# B&R Automation Studio project GAT (part 8)

#### Configuration.st - not listed in the package file held
```iecst
ACTION ConfigurationInit:

    MachineSettings.DriveConfiguration.PureVirtualAxis.AxisFeatures.FeatureReference.DataAddress := ADR(MachineSettings.AxisFeatures);
    MachineSettings.DriveConfiguration.PureVirtualAxis.AxisFeatures.FeatureReference.NumberOfArrayElements := SIZEOF(MachineSettings.AxisFeatures)/SIZEOF(MachineSettings.AxisFeatures[0]);
    MachineSettings.DriveConfiguration.PureVirtualAxis.AxisFeatures.FeatureReference.NumberOfElements := 0;
    i := 0;
    WHILE ((i <= SIZEOF(MachineSettings.AxisFeatures)/SIZEOF(MachineSettings.AxisFeatures[0])) AND (MachineSettings.AxisFeatures[i] <> '')) DO
        i := i + 1;
    END_WHILE
    MachineSettings.DriveConfiguration.PureVirtualAxis.AxisFeatures.FeatureReference.NumberOfElements := i;

    MC_BR_ProcessConfig_AX.DataAddress := ADR(MachineSettings.BaseConfiguration);
    MC_BR_ProcessConfig_AX.DataType := mcCFG_AX;

    MC_BR_ProcessConfig_ACP.DataAddress := ADR(MachineSettings.DriveConfiguration);
    MC_BR_ProcessConfig_ACP.DataType := mcCFG_PURE_V_AX;

    configurationState := CONFIG_STATE_INIT;

END_ACTION

ACTION Configuration:

    CASE configurationState OF
        CONFIG_STATE_INIT:

            (* build up the string for the name *)
            MC_BR_ProcessConfig_ACP.Name := MpAxisBasicFB.Info.HardwareInfo.Axis.ConfigElementLocation;
            MC_BR_ProcessConfig_AX.Name := MpAxisBasicFB.Info.HardwareInfo.Axis.AxisName;

            IF (MpAxisBasicFB.Active = TRUE) THEN
                configurationState := CONFIG_STATE_READ;
            END_IF

        CONFIG_STATE_READ:
            MC_BR_ProcessConfig_ACP.Mode := mcPCM_LOAD;
            MC_BR_ProcessConfig_ACP.Execute := TRUE;

            MC_BR_ProcessConfig_AX.Mode := mcPCM_LOAD;
            MC_BR_ProcessConfig_AX.Execute := TRUE;
            IF (MC_BR_ProcessConfig_ACP.Done = TRUE) AND (MC_BR_ProcessConfig_AX.Done = TRUE) THEN
                MC_BR_ProcessConfig_ACP.Execute := FALSE;
                MC_BR_ProcessConfig_AX.Execute := FALSE;
                configurationState := CONFIG_STATE_READY;
            END_IF

        CONFIG_STATE_WRITE:
            MC_BR_ProcessConfig_ACP.Mode := mcPCM_SAVE;
            MC_BR_ProcessConfig_ACP.Execute := TRUE;

            MC_BR_ProcessConfig_AX.Mode := mcPCM_SAVE;
            MC_BR_ProcessConfig_AX.Execute := TRUE;
            IF (MC_BR_ProcessConfig_ACP.Done = TRUE) AND (MC_BR_ProcessConfig_AX.Done = TRUE) THEN
                MC_BR_ProcessConfig_ACP.Execute := FALSE;
                MC_BR_ProcessConfig_AX.Execute := FALSE;
                configurationState := CONFIG_STATE_READY;
            END_IF

        CONFIG_STATE_READY:

    END_CASE

    MC_BR_ProcessConfig_ACP();
    MC_BR_ProcessConfig_AX();

END_ACTION
```

#### Main.st - not listed in the package file held
```iecst
(***********************************************************************************************************************
* Copyright: B&R Industrial Automation GmbH
* Description: This program implements an axis control
***********************************************************************************************************************)

PROGRAM _INIT

    ST_name(0, ADR(AxisControl.Status.TaskName), 0);

    MpAlarmXCoreFB.Enable := TRUE;
    ConfigurationInit;

    MpAxisBasicFB.Enable := TRUE;
    MpAxisBasicFB.MpLink := ADR(gAxisTest);

    AxisInit;

END_PROGRAM

PROGRAM _CYCLIC

    MpAxisBasicFB.MpLink := ADR(gAxisTest);
    MC_BR_CheckRestorePositionDataFB.Axis := ADR(gAxisTest);

    SimulationControl;
    AxisStateMachine;
    AxisCyclic;
    RecipeCyclic;

    MpAlarmXCoreFB.MpLink := ADR(gAlarmXCore_Test);
    MpAlarmXCoreFB();

END_PROGRAM

PROGRAM _EXIT

    MpRecipeRegPar_MachineFB.Enable := FALSE;
    MpRecipeRegPar_MachineFB();

    MpRecipeRegPar_UserFB.Enable := FALSE;
    MpRecipeRegPar_UserFB();

    MpRecipeRegPar_PreFB.Enable := FALSE;
    MpRecipeRegPar_PreFB();

    MpRecipeRegPar_UserPreFB.Enable := FALSE;
    MpRecipeRegPar_UserPreFB();

    MpAxisBasicFB.Enable := FALSE;
    MpAxisBasicFB();

    MpAlarmXCoreFB.Enable := FALSE;
    MpAlarmXCoreFB();

END_PROGRAM
```

### Program Logical/Infrastructure/UsbDevLink/UsbDevLink (IEC)

#### UsbDevLink.st - Init, cyclic, exit code
```iecst
//*********************************************************************************
//* Copyright: B&R Industrial Automation GmbH
//* Author:    MITC
//* Created:   September 26, 2021/09:19
//* This task shall automatically detect and (un)link USB storage devices
//*********************************************************************************

PROGRAM _INIT
	DevLinkCtrl.FUB.DevLink_0.enable := FALSE;
	DevLinkCtrl.FUB.DevUnlink_0.enable := FALSE;
	DevLinkCtrl.FUB.UsbNodeGet_0.enable := FALSE;
	DevLinkCtrl.FUB.UsbNodeListGet_0.enable := FALSE;
	DevLinkCtrl.FUB.DevLink_0();
	DevLinkCtrl.FUB.DevUnlink_0();
	DevLinkCtrl.FUB.UsbNodeGet_0();
	DevLinkCtrl.FUB.UsbNodeListGet_0();

	FOR Index := 0 TO MAX_IDX_USB_DEV_LIST DO
		AttachedUSB[Index] := FALSE;
		gUSBAvailable[Index] := FALSE;
	END_FOR
END_PROGRAM

PROGRAM _CYCLIC
	// BEGIN OF STATE MACHINE
	CASE DevLinkCtrl.Step OF
		// WAIT STEP
		STATE_WAIT:
			// UPDATE USB INFO LIST IF THE NODE LIST HAS CHANGED
			IF (brsmemcmp(ADR(DevLinkCtrl.Params.NodeList), ADR(LastNodeList), SIZEOF(LastNodeList)) <> 0) THEN
				DevLinkCtrl.Cmd.GetUSBInfo := TRUE;
				// preserve the previously created drive information in CASE the order has changed when unplugging a device
				FOR DevLinkCtrl.Params.Index := 0 TO MAX_IDX_USB_DEV_LIST DO
					FOR Index := 0 TO MAX_IDX_USB_DEV_LIST DO
						IF ((DevLinkCtrl.Params.NodeList[DevLinkCtrl.Params.Index] = LastNodeList[Index]) AND
							(DevLinkCtrl.Params.Index <> Index) AND (LastNodeList[Index] <> 0)) THEN
							brsmemcpy(ADR(TempUSBInfo), ADR(DevLinkCtrl.Params.NodeInfoList[DevLinkCtrl.Params.Index]), SIZEOF(TempUSBInfo));
							brsmemcpy(ADR(DevLinkCtrl.Params.NodeInfoList[DevLinkCtrl.Params.Index]), ADR(DevLinkCtrl.Params.NodeInfoList[Index]), SIZEOF(TempUSBInfo));
							brsmemcpy(ADR(DevLinkCtrl.Params.NodeInfoList[Index]), ADR(TempUSBInfo), SIZEOF(TempUSBInfo));
							brsmemcpy(ADR(TempFileDevName), ADR(DevLinkCtrl.Params.FileDevName[DevLinkCtrl.Params.Index]), SIZEOF(TempFileDevName));
							brsmemcpy(ADR(DevLinkCtrl.Params.FileDevName[DevLinkCtrl.Params.Index]), ADR(DevLinkCtrl.Params.FileDevName[Index]), SIZEOF(TempFileDevName));
							brsmemcpy(ADR(DevLinkCtrl.Params.FileDevName[Index]), ADR(TempFileDevName), SIZEOF(TempFileDevName));
							TempFileDevHandle := DevLinkCtrl.Params.FileDevHandle[DevLinkCtrl.Params.Index];
							DevLinkCtrl.Params.FileDevHandle[DevLinkCtrl.Params.Index] := DevLinkCtrl.Params.FileDevHandle[Index];
							DevLinkCtrl.Params.FileDevHandle[Index] := TempFileDevHandle;
						END_IF
					END_FOR
				END_FOR
				brsmemcpy(ADR(LastNodeList), ADR(DevLinkCtrl.Params.NodeList), SIZEOF(LastNodeList));
			END_IF

			FOR DevLinkCtrl.Params.Index := 0 TO MAX_IDX_USB_DEV_LIST DO
				// SKIP IF LOADING USB LIST INFORMATION
				IF DevLinkCtrl.Cmd.GetUSBInfo THEN
					EXIT;
				END_IF
				// ALWAYS KEEP DEVICES LINKED WHEN AVAILABLE
				IF ((DevLinkCtrl.Params.FileDevHandle[DevLinkCtrl.Params.Index] = 0) AND AttachedUSB[DevLinkCtrl.Params.Index]
					AND (DevLinkCtrl.Params.NodeList[DevLinkCtrl.Params.Index] <> 0)) THEN
					DevLinkCtrl.Cmd.DevLink := TRUE;
					EXIT;
				END_IF
				// UNLINK DEVICE IF IT IS NOT CONNECTED ANYMORE
				IF ((DevLinkCtrl.Params.FileDevHandle[DevLinkCtrl.Params.Index] <> 0) AND
					(DevLinkCtrl.Params.NodeInfoList[DevLinkCtrl.Params.Index].interfaceClass <> 8)) THEN
					DevLinkCtrl.Cmd.DevUnlink := TRUE;
					EXIT;
				END_IF
			END_FOR

			// CHECK FOR USB DEVICES EVERY 3 SEC
			TON_0.PT := t#3s;
			IF (TON_0.Q AND NOT DevLinkCtrl.Cmd.GetUSBInfo AND NOT DevLinkCtrl.Cmd.DevLink AND NOT DevLinkCtrl.Cmd.DevUnlink) THEN
				DevLinkCtrl.Cmd.GetUSBList := TRUE;
				TON_0.IN := FALSE;
			ELSE
				TON_0.IN := TRUE;
			END_IF
			TON_0();

			IF DevLinkCtrl.Cmd.GetUSBInfo THEN
				// get usb info cmd
				DevLinkCtrl.Cmd.GetUSBInfo := FALSE;
				brsmemset(ADR(DevLinkCtrl.Params.NodeInfoList), 0, SIZEOF(DevLinkCtrl.Params.NodeInfoList));
				DevLinkCtrl.Step := STATE_GET_USB_INFO;
				DevLinkCtrl.Params.Index := 0;
			ELSIF DevLinkCtrl.Cmd.GetUSBList THEN
				// get usb list cmd
				DevLinkCtrl.Cmd.GetUSBList := FALSE;
				brsmemset(ADR(DevLinkCtrl.Params.NodeList), 0, SIZEOF(DevLinkCtrl.Params.NodeList));
				DevLinkCtrl.Step := STATE_GET_USB_LIST;
			ELSIF DevLinkCtrl.Cmd.DevLink THEN
				// link cmd
				DevLinkCtrl.Cmd.DevLink := FALSE;
				DevLinkCtrl.Step := STATE_DEV_LINK;
			ELSIF DevLinkCtrl.Cmd.DevUnlink THEN
				// unlink cmd
				DevLinkCtrl.Cmd.DevUnlink := FALSE;
				DevLinkCtrl.Step := STATE_DEV_UNLINK;
			END_IF
			// END OF WAIT STEP

			// GET USB LIST STEP
		STATE_GET_USB_LIST:
			// SET FUB PARAMS
			DevLinkCtrl.FUB.UsbNodeListGet_0.enable := TRUE;
			DevLinkCtrl.FUB.UsbNodeListGet_0.bufferSize := SIZEOF(DevLinkCtrl.Params.NodeList);
			DevLinkCtrl.FUB.UsbNodeListGet_0.pBuffer := ADR(DevLinkCtrl.Params.NodeList);

			// ERROR HANDLING
			IF ((DevLinkCtrl.FUB.UsbNodeListGet_0.status = ERR_OK) OR (DevLinkCtrl.FUB.UsbNodeListGet_0.status = asusbERR_USB_NOTFOUND)) THEN
				DevLinkCtrl.Step := STATE_WAIT;
				DevLinkCtrl.FUB.UsbNodeListGet_0.enable := FALSE;
			ELSIF ((DevLinkCtrl.FUB.UsbNodeListGet_0.status <> ERR_FUB_BUSY) AND (DevLinkCtrl.FUB.UsbNodeListGet_0.status <> ERR_FUB_ENABLE_FALSE)
				AND (DevLinkCtrl.FUB.UsbNodeListGet_0.status <> asusbERR_USB_NOTFOUND)) THEN
				DevLinkCtrl.Step := STATE_ERROR_USB;
				DevLinkCtrl.Params.ErrorID := DevLinkCtrl.FUB.UsbNodeListGet_0.status;
				DevLinkCtrl.FUB.UsbNodeListGet_0.enable := FALSE;
			END_IF
			// CALL OF FUB
			DevLinkCtrl.FUB.UsbNodeListGet_0();
			// END OF GET USB LIST STEP

			// GET USB INFO STEP
		STATE_GET_USB_INFO:
			// SET FUB PARAMS
			DevLinkCtrl.FUB.UsbNodeGet_0.bufferSize := SIZEOF(DevLinkCtrl.Params.NodeInfoList[DevLinkCtrl.Params.Index]);
			DevLinkCtrl.FUB.UsbNodeGet_0.enable := TRUE;
			DevLinkCtrl.FUB.UsbNodeGet_0.nodeId := DevLinkCtrl.Params.NodeList[DevLinkCtrl.Params.Index];
			DevLinkCtrl.FUB.UsbNodeGet_0.pBuffer := ADR(DevLinkCtrl.Params.NodeInfoList[DevLinkCtrl.Params.Index]);

			// CHECK IF DevLinkCtrl.Params.Index CONTAINS AN ENTRY
			IF (DevLinkCtrl.Params.NodeList[DevLinkCtrl.Params.Index] = 0) THEN
				DevLinkCtrl.FUB.UsbNodeGet_0.enable := TRUE;
				brsmemset(ADR(DevLinkCtrl.Params.NodeInfoList[DevLinkCtrl.Params.Index]), 0, SIZEOF(DevLinkCtrl.Params.NodeInfoList[DevLinkCtrl.Params.Index]));
				DevLinkCtrl.Params.Index := DevLinkCtrl.Params.Index + 1;
			END_IF

			// ERROR HANDLING
			IF (DevLinkCtrl.FUB.UsbNodeGet_0.status = ERR_OK) THEN
				DevLinkCtrl.FUB.UsbNodeGet_0.enable := FALSE;
				DevLinkCtrl.Params.Index := DevLinkCtrl.Params.Index + 1;
			ELSIF ((DevLinkCtrl.FUB.UsbNodeGet_0.status <> ERR_FUB_BUSY) AND (DevLinkCtrl.FUB.UsbNodeGet_0.status <> ERR_FUB_ENABLE_FALSE)) THEN
				DevLinkCtrl.Step := STATE_ERROR_USB;
				DevLinkCtrl.Params.ErrorID := DevLinkCtrl.FUB.UsbNodeGet_0.status;
				DevLinkCtrl.FUB.UsbNodeGet_0.enable := FALSE;
			END_IF

			// END OF LIST REACHED
			IF (DevLinkCtrl.Params.Index > MAX_IDX_USB_DEV_LIST) THEN
				DevLinkCtrl.FUB.UsbNodeGet_0.enable := FALSE;
				DevLinkCtrl.Step := STATE_WAIT;
				FOR DevLinkCtrl.Params.Index := 0 TO MAX_IDX_USB_DEV_LIST DO
					IF (DevLinkCtrl.Params.NodeInfoList[DevLinkCtrl.Params.Index].interfaceClass = 8) THEN
						AttachedUSB[DevLinkCtrl.Params.Index] := TRUE;
					ELSE
						AttachedUSB[DevLinkCtrl.Params.Index] := FALSE;
						gUSBAvailable[DevLinkCtrl.Params.Index] := FALSE;
					END_IF
				END_FOR
			END_IF

			// CALL OF FUB
			DevLinkCtrl.FUB.UsbNodeGet_0();
			// END OF GET USB INFO STEP

			// LINK DEVICE STEP
		STATE_DEV_LINK:
            // SET FUB PARAMS
			DevLinkCtrl.FUB.DevLink_0.enable := TRUE;
			DevLinkCtrl.FUB.DevLink_0.pDevice := ADR(DevLinkCtrl.Params.FileDevName[DevLinkCtrl.Params.Index]);
			brsstrcpy(ADR(DevLinkCtrl.Params.LinkParam), ADR('/DEVICE='));
			brsstrcat(ADR(DevLinkCtrl.Params.LinkParam), ADR(DevLinkCtrl.Params.NodeInfoList[DevLinkCtrl.Params.Index].ifName));
			DevLinkCtrl.FUB.DevLink_0.pParam := ADR(DevLinkCtrl.Params.LinkParam);

			// ERROR HANDLING
			IF (DevLinkCtrl.FUB.DevLink_0.status = ERR_OK) THEN
				DevLinkCtrl.Params.FileDevHandle[DevLinkCtrl.Params.Index] := DevLinkCtrl.FUB.DevLink_0.handle;
				DevLinkCtrl.Step := STATE_WAIT;
				DevLinkCtrl.FUB.DevLink_0.enable := FALSE;
				FOR Index := 0 TO MAX_IDX_USB_DEV_LIST DO
					gUSBAvailable[Index] := AttachedUSB[Index];
				END_FOR
			ELSIF ((DevLinkCtrl.FUB.DevLink_0.status <> ERR_FUB_BUSY) AND (DevLinkCtrl.FUB.DevLink_0.status <> ERR_FUB_ENABLE_FALSE)) THEN
				DevLinkCtrl.Step := STATE_ERROR_USB;
				DevLinkCtrl.Params.ErrorID := DevLinkCtrl.FUB.DevLink_0.status;
				DevLinkCtrl.FUB.DevLink_0.enable := FALSE;
			END_IF
			// CALL OF FUB
			DevLinkCtrl.FUB.DevLink_0();
			// END OF LINK DEVICE STEP

			// UNLINK DEVICE STEP
		STATE_DEV_UNLINK:
			// SET FUB PARAMS
			DevLinkCtrl.FUB.DevUnlink_0.enable := TRUE;
			DevLinkCtrl.FUB.DevUnlink_0.handle := DevLinkCtrl.Params.FileDevHandle[DevLinkCtrl.Params.Index];

			// CHECK IF WE HAVE A HANDLE
			IF (DevLinkCtrl.Params.FileDevHandle[DevLinkCtrl.Params.Index] = 0) THEN
				DevLinkCtrl.FUB.DevUnlink_0.enable := FALSE;
				DevLinkCtrl.Step := STATE_WAIT;
			END_IF

			// ERROR HANDLING
			IF (DevLinkCtrl.FUB.DevUnlink_0.status = ERR_OK) THEN
				DevLinkCtrl.Params.FileDevHandle[DevLinkCtrl.Params.Index] := 0;
				DevLinkCtrl.FUB.DevUnlink_0.enable := FALSE;
				DevLinkCtrl.Step := STATE_WAIT;
			ELSIF ((DevLinkCtrl.FUB.DevUnlink_0.status <> ERR_FUB_BUSY) AND (DevLinkCtrl.FUB.DevUnlink_0.status <> ERR_FUB_ENABLE_FALSE)) THEN
				DevLinkCtrl.Step := STATE_ERROR_USB;
				DevLinkCtrl.Params.ErrorID := DevLinkCtrl.FUB.DevUnlink_0.status;
				DevLinkCtrl.FUB.DevUnlink_0.enable := FALSE;
			END_IF
			// CALL OF FUB
			DevLinkCtrl.FUB.DevUnlink_0();
			// END OF UNLINK DEVICE STEP

			// WAIT FOR ERRACK CMD STEP
		STATE_ERROR_USB:
			// DELETE ERROR ID AND GO BACK TO WAIT STEP WHEN ERROR IS ACKNOWLEDGED
			IF DevLinkCtrl.Cmd.ErrAck THEN
				DevLinkCtrl.Params.ErrorID := 0;
				DevLinkCtrl.Cmd.ErrAck := FALSE;
				DevLinkCtrl.Step := STATE_WAIT;
			END_IF
		// END OF WAIT FOR ERRACK STEP
	END_CASE;
	// END OF STATE MACHINE
END_PROGRAM

PROGRAM _EXIT
	// Insert code here
END_PROGRAM
```

#### UsbDevLink.var - Local variables
```iecst
(*********************************************************************************
 * Copyright: Bernecker + Rainer
 * Author:    deermannd
 * Created:   21 October, 2015/1:30 PM
 *********************************************************************************
 * DevLinkTask variables of project
 *********************************************************************************)
VAR
	DevLinkCtrl : DevLinkCtrlType := (Params:=(FileDevName:=['USB1','USB2'])); (*DevLink Control variable*)
	TON_0 : TON; (*timer to refresh available usb devices*)
	LastNodeList : ARRAY[0..MAX_IDX_USB_DEV_LIST] OF UDINT; (*temp variable to check if the node list has changed*)
	TempFileDevHandle : UDINT := 0;
	TempFileDevName : STRING[30] := '';
	TempUSBInfo : usbNode_typ := (0); (*temp info structure*)
	Index : USINT := 0; (*index to loop through ussb devices*)
	AttachedUSB : ARRAY[0..MAX_IDX_USB_DEV_LIST] OF BOOL := [2(FALSE)];
END_VAR
```

#### Types.typ - not listed in the package file held
```iecst
(*********************************************************************************
 * Copyright: Bernecker + Rainer
 * Author:    MITC
 * Created:   21 October, 2015/1:30 PM
 *********************************************************************************
 * DevLinkTask data types of project
 *********************************************************************************)

TYPE
	StepType :
		( (*enumeration of the possible machine states*)
		STATE_WAIT := 0, (*waiting for cmds*)
		STATE_GET_USB_LIST, (*getting list of usb devices*)
		STATE_GET_USB_INFO, (*getting info from a usb device*)
		STATE_DEV_LINK, (*linking device*)
		STATE_DEV_UNLINK, (*unlinking device*)
		STATE_ERROR_USB (*some FUB returned an error*)
		);
	CommandType : 	STRUCT  (*possible machine cmds*)
		GetUSBList : BOOL; (*get usb list cmd*)
		GetUSBInfo : BOOL; (*get usb info cmd*)
		DevLink : BOOL; (*link cmd*)
		DevUnlink : BOOL; (*unlink cmd*)
		ErrAck : BOOL; (*error acknowledge cmd*)
	END_STRUCT;
	DevLink_FUB_Type : 	STRUCT  (*contains all needed FileIO FUBs*)
		UsbNodeListGet_0 : UsbNodeListGet;
		UsbNodeGet_0 : UsbNodeGet;
		UsbMsDeviceReady_0 : UsbMsDeviceReady;
		DevLink_0 : DevLink;
		DevUnlink_0 : DevUnlink;
	END_STRUCT;
	DevLinkCtrlType : 	STRUCT  (*Control structure which contains everything necessary for the file handling machine*)
		Step : StepType; (*actual step*)
		Cmd : CommandType; (*when in STATE_WAIT a cmd with value true will change the machine state*)
		FUB : DevLink_FUB_Type; (*all DevLink FUBs*)
		Params : ParamsType; (*parameters like file device, error ID, Buffer, ...*)
	END_STRUCT;
	ParamsType : 	STRUCT  (*Parameter structure*)
		ErrorID : UINT; (*the error id from a FUB is stored here in case of error*)
		NodeList : ARRAY[0..MAX_IDX_USB_DEV_LIST]OF UDINT; (*List of connected usb devices*)
		NodeInfoList : ARRAY[0..MAX_IDX_USB_DEV_LIST]OF usbNode_typ; (*Buffer for usb info*)
		FileDevName : ARRAY[0..MAX_IDX_USB_DEV_LIST]OF STRING[30]; (*file device names*)
		FileDevHandle : ARRAY[0..MAX_IDX_USB_DEV_LIST]OF UDINT; (*needed for unlinking the device again*)
		LinkParam : STRING[30]; (*param string to link a device*)
		Index : USINT; (*list index*)
	END_STRUCT;
END_TYPE
```

#### Variables.var - not listed in the package file held
```iecst
(*********************************************************************************
 * Copyright: Bernecker + Rainer
 * Author:    deermannd
 * Created:   21 October, 2015/1:30 PM
 *********************************************************************************
 * DevLinkTask variables of project
 *********************************************************************************)
VAR CONSTANT
	MAX_IDX_USB_DEV_LIST : USINT := 1; (*Max index for usb storage devices (1 means up to two devices with index 0 and 1)*)
END_VAR
VAR
	DevLinkCtrl : DevLinkCtrlType := (Params:=(FileDevName:=['USB1','USB2'])); (*DevLink Control variable*)
	TON_0 : TON; (*timer to refresh available usb devices*)
	LastNodeList : ARRAY[0..MAX_IDX_USB_DEV_LIST] OF UDINT; (*temp variable to check if the node list has changed*)
	TempFileDevHandle : UDINT := 0;
	TempFileDevName : STRING[30] := '';
	TempUSBInfo : usbNode_typ := (0); (*temp info structure*)
	Index : USINT := 0; (*index to loop through ussb devices*)
	bAttachedUSB : ARRAY[0..MAX_IDX_USB_DEV_LIST] OF BOOL := [2(FALSE)];
END_VAR
```

#### Main.st - not listed in the package file held
```iecst
(*********************************************************************************
 * Copyright: B&R Industrial Automation GmbH
 * Author:    MITC
 * Created:   September 26, 2021/09:19
 * This task shall automatically detect and (un)link USB storage devices
 *********************************************************************************)

PROGRAM _INIT
	DevLinkCtrl.FUB.DevLink_0.enable		:= FALSE;
	DevLinkCtrl.FUB.DevUnlink_0.enable 		:= FALSE;
	DevLinkCtrl.FUB.UsbNodeGet_0.enable		:= FALSE;
	DevLinkCtrl.FUB.UsbNodeListGet_0.enable	:= FALSE;
	DevLinkCtrl.FUB.DevLink_0();
	DevLinkCtrl.FUB.DevUnlink_0();
	DevLinkCtrl.FUB.UsbNodeGet_0();
	DevLinkCtrl.FUB.UsbNodeListGet_0();

	FOR Index := 0 TO MAX_IDX_USB_DEV_LIST DO
		bAttachedUSB[Index] 				:= FALSE;
		gbUSBAvail[Index]					:= FALSE;
	END_FOR;
END_PROGRAM

PROGRAM _CYCLIC
	(* BEGIN OF STATE MACHINE *)
	CASE DevLinkCtrl.Step OF
		(* WAIT STEP *)
		STATE_WAIT:
			(* UPDATE USB INFO LIST IF THE NODE LIST HAS CHANGED *)
			IF (brsmemcmp(ADR(DevLinkCtrl.Params.NodeList), ADR(LastNodeList), SIZEOF(LastNodeList)) <> 0) THEN
				DevLinkCtrl.Cmd.GetUSBInfo		:= TRUE;
				(* preserve the previously created drive information in CASE the order has changed when unplugging a device *)
				FOR DevLinkCtrl.Params.Index := 0 TO MAX_IDX_USB_DEV_LIST DO
					FOR Index := 0 TO MAX_IDX_USB_DEV_LIST DO
						IF ((DevLinkCtrl.Params.NodeList[DevLinkCtrl.Params.Index] = LastNodeList[Index]) AND
							(DevLinkCtrl.Params.Index <> Index) AND (LastNodeList[Index] <> 0)) THEN
							brsmemcpy(ADR(TempUSBInfo), ADR(DevLinkCtrl.Params.NodeInfoList[DevLinkCtrl.Params.Index]), SIZEOF(TempUSBInfo));
							brsmemcpy(ADR(DevLinkCtrl.Params.NodeInfoList[DevLinkCtrl.Params.Index]), ADR(DevLinkCtrl.Params.NodeInfoList[Index]), SIZEOF(TempUSBInfo));
							brsmemcpy(ADR(DevLinkCtrl.Params.NodeInfoList[Index]), ADR(TempUSBInfo), SIZEOF(TempUSBInfo));
							brsmemcpy(ADR(TempFileDevName), ADR(DevLinkCtrl.Params.FileDevName[DevLinkCtrl.Params.Index]), SIZEOF(TempFileDevName));
							brsmemcpy(ADR(DevLinkCtrl.Params.FileDevName[DevLinkCtrl.Params.Index]), ADR(DevLinkCtrl.Params.FileDevName[Index]), SIZEOF(TempFileDevName));
							brsmemcpy(ADR(DevLinkCtrl.Params.FileDevName[Index]), ADR(TempFileDevName), SIZEOF(TempFileDevName));
							TempFileDevHandle											:= DevLinkCtrl.Params.FileDevHandle[DevLinkCtrl.Params.Index];
							DevLinkCtrl.Params.FileDevHandle[DevLinkCtrl.Params.Index]	:= DevLinkCtrl.Params.FileDevHandle[Index];
							DevLinkCtrl.Params.FileDevHandle[Index]						:= TempFileDevHandle;
						END_IF;
					END_FOR;
				END_FOR;
				brsmemcpy(ADR(LastNodeList), ADR(DevLinkCtrl.Params.NodeList), SIZEOF(LastNodeList));
			END_IF;

			FOR DevLinkCtrl.Params.Index := 0 TO MAX_IDX_USB_DEV_LIST DO
				(* SKIP IF LOADING USB LIST INFORMATION *)
				IF DevLinkCtrl.Cmd.GetUSBInfo THEN
					EXIT;
				END_IF;
				(* ALWAYS KEEP DEVICES LINKED WHEN AVAILABLE *)
				IF ((DevLinkCtrl.Params.FileDevHandle[DevLinkCtrl.Params.Index] = 0) AND bAttachedUSB[DevLinkCtrl.Params.Index]
					AND (DevLinkCtrl.Params.NodeList[DevLinkCtrl.Params.Index] <> 0)) THEN
					DevLinkCtrl.Cmd.DevLink		:= TRUE;
					EXIT;
				END_IF;
				(* UNLINK DEVICE IF IT IS NOT CONNECTED ANYMORE *)
				IF ((DevLinkCtrl.Params.FileDevHandle[DevLinkCtrl.Params.Index] <> 0) AND
					(DevLinkCtrl.Params.NodeInfoList[DevLinkCtrl.Params.Index].interfaceClass <> 8)) THEN
					DevLinkCtrl.Cmd.DevUnlink	:= TRUE;
					EXIT;
				END_IF;
			END_FOR;

			(* CHECK FOR USB DEVICES EVERY 3 SEC *)
			TON_0.PT							:= t#3s;
			IF (TON_0.Q AND NOT DevLinkCtrl.Cmd.GetUSBInfo AND NOT DevLinkCtrl.Cmd.DevLink AND NOT DevLinkCtrl.Cmd.DevUnlink) THEN
				DevLinkCtrl.Cmd.GetUSBList		:= TRUE;
				TON_0.IN						:= FALSE;
			ELSE
				TON_0.IN						:= TRUE;
			END_IF;
			TON_0();

			IF DevLinkCtrl.Cmd.GetUSBInfo THEN
				(* get usb info cmd *)
				DevLinkCtrl.Cmd.GetUSBInfo	:= FALSE;
				brsmemset(ADR(DevLinkCtrl.Params.NodeInfoList), 0, SIZEOF(DevLinkCtrl.Params.NodeInfoList));
				DevLinkCtrl.Step			:= STATE_GET_USB_INFO;
				DevLinkCtrl.Params.Index	:= 0;
			ELSIF DevLinkCtrl.Cmd.GetUSBList THEN
				(* get usb list cmd *)
				DevLinkCtrl.Cmd.GetUSBList	:= FALSE;
				brsmemset(ADR(DevLinkCtrl.Params.NodeList), 0, SIZEOF(DevLinkCtrl.Params.NodeList));
				DevLinkCtrl.Step			:= STATE_GET_USB_LIST;
			ELSIF DevLinkCtrl.Cmd.DevLink THEN
				(* link cmd *)
				DevLinkCtrl.Cmd.DevLink		:= FALSE;
				DevLinkCtrl.Step			:= STATE_DEV_LINK;
			ELSIF DevLinkCtrl.Cmd.DevUnlink THEN
				(* unlink cmd *)
				DevLinkCtrl.Cmd.DevUnlink	:= FALSE;
				DevLinkCtrl.Step			:= STATE_DEV_UNLINK;
			END_IF;
			(* END OF WAIT STEP *)

			(* GET USB LIST STEP *)
		STATE_GET_USB_LIST:
			(* SET FUB PARAMS *)
			DevLinkCtrl.FUB.UsbNodeListGet_0.enable		:= TRUE;
			DevLinkCtrl.FUB.UsbNodeListGet_0.bufferSize	:= SIZEOF(DevLinkCtrl.Params.NodeList);
			DevLinkCtrl.FUB.UsbNodeListGet_0.pBuffer	:= ADR(DevLinkCtrl.Params.NodeList);

			(* ERROR HANDLING *)
			IF ((DevLinkCtrl.FUB.UsbNodeListGet_0.status = ERR_OK) OR (DevLinkCtrl.FUB.UsbNodeListGet_0.status = asusbERR_USB_NOTFOUND)) THEN
				DevLinkCtrl.Step						:= STATE_WAIT;
				DevLinkCtrl.FUB.UsbNodeListGet_0.enable	:= FALSE;
			ELSIF ((DevLinkCtrl.FUB.UsbNodeListGet_0.status <> ERR_FUB_BUSY) AND (DevLinkCtrl.FUB.UsbNodeListGet_0.status <> ERR_FUB_ENABLE_FALSE)
				AND (DevLinkCtrl.FUB.UsbNodeListGet_0.status <> asusbERR_USB_NOTFOUND)) THEN
				DevLinkCtrl.Step						:= STATE_ERROR_USB;
				DevLinkCtrl.Params.ErrorID				:= DevLinkCtrl.FUB.UsbNodeListGet_0.status;
				DevLinkCtrl.FUB.UsbNodeListGet_0.enable	:= FALSE;
			END_IF;
			(* CALL OF FUB *)
			DevLinkCtrl.FUB.UsbNodeListGet_0();
			(* END OF GET USB LIST STEP *)

			(* GET USB INFO STEP *)
		STATE_GET_USB_INFO:
			(* SET FUB PARAMS *)
			DevLinkCtrl.FUB.UsbNodeGet_0.bufferSize	:= SIZEOF(DevLinkCtrl.Params.NodeInfoList[DevLinkCtrl.Params.Index]);
			DevLinkCtrl.FUB.UsbNodeGet_0.enable		:= TRUE;
			DevLinkCtrl.FUB.UsbNodeGet_0.nodeId		:= DevLinkCtrl.Params.NodeList[DevLinkCtrl.Params.Index];
			DevLinkCtrl.FUB.UsbNodeGet_0.pBuffer	:= ADR(DevLinkCtrl.Params.NodeInfoList[DevLinkCtrl.Params.Index]);

			(* CHECK IF DevLinkCtrl.Params.Index CONTAINS AN ENTRY *)
			IF (DevLinkCtrl.Params.NodeList[DevLinkCtrl.Params.Index] = 0) THEN
				DevLinkCtrl.FUB.UsbNodeGet_0.enable	:= TRUE;
				brsmemset(ADR(DevLinkCtrl.Params.NodeInfoList[DevLinkCtrl.Params.Index]), 0, SIZEOF(DevLinkCtrl.Params.NodeInfoList[DevLinkCtrl.Params.Index]));
				DevLinkCtrl.Params.Index			:= DevLinkCtrl.Params.Index + 1;
			END_IF;

			(* ERROR HANDLING *)
			IF (DevLinkCtrl.FUB.UsbNodeGet_0.status = ERR_OK) THEN
				DevLinkCtrl.FUB.UsbNodeGet_0.enable	:= FALSE;
				DevLinkCtrl.Params.Index			:= DevLinkCtrl.Params.Index + 1;
			ELSIF ((DevLinkCtrl.FUB.UsbNodeGet_0.status <> ERR_FUB_BUSY) AND (DevLinkCtrl.FUB.UsbNodeGet_0.status <> ERR_FUB_ENABLE_FALSE)) THEN
				DevLinkCtrl.Step					:= STATE_ERROR_USB;
				DevLinkCtrl.Params.ErrorID			:= DevLinkCtrl.FUB.UsbNodeGet_0.status;
				DevLinkCtrl.FUB.UsbNodeGet_0.enable	:= FALSE;
			END_IF;

			(* END OF LIST REACHED *)
			IF (DevLinkCtrl.Params.Index > MAX_IDX_USB_DEV_LIST) THEN
				DevLinkCtrl.FUB.UsbNodeGet_0.enable	:= FALSE;
				DevLinkCtrl.Step					:= STATE_WAIT;
				FOR DevLinkCtrl.Params.Index := 0 TO MAX_IDX_USB_DEV_LIST DO
					IF (DevLinkCtrl.Params.NodeInfoList[DevLinkCtrl.Params.Index].interfaceClass = 8) THEN
						bAttachedUSB[DevLinkCtrl.Params.Index]	:= TRUE;
					ELSE
						bAttachedUSB[DevLinkCtrl.Params.Index]	:= FALSE;
						gbUSBAvail[DevLinkCtrl.Params.Index]	:= FALSE;
					END_IF;
				END_FOR;
			END_IF;

			(* CALL OF FUB *)
			DevLinkCtrl.FUB.UsbNodeGet_0();
			(* END OF GET USB INFO STEP *)

			(* LINK DEVICE STEP *)
		STATE_DEV_LINK:
			(* SET FUB PARAMS *)
			DevLinkCtrl.FUB.DevLink_0.enable	:= TRUE;
			DevLinkCtrl.FUB.DevLink_0.pDevice	:= ADR(DevLinkCtrl.Params.FileDevName[DevLinkCtrl.Params.Index]);
			brsstrcpy(ADR(DevLinkCtrl.Params.LinkParam), ADR('/DEVICE='));
			brsstrcat(ADR(DevLinkCtrl.Params.LinkParam), ADR(DevLinkCtrl.Params.NodeInfoList[DevLinkCtrl.Params.Index].ifName));
			DevLinkCtrl.FUB.DevLink_0.pParam	:= ADR(DevLinkCtrl.Params.LinkParam);

			(* ERROR HANDLING *)
			IF (DevLinkCtrl.FUB.DevLink_0.status = ERR_OK) THEN
				DevLinkCtrl.Params.FileDevHandle[DevLinkCtrl.Params.Index]	:= DevLinkCtrl.FUB.DevLink_0.handle;
				DevLinkCtrl.Step											:= STATE_WAIT;
				DevLinkCtrl.FUB.DevLink_0.enable							:= FALSE;
				FOR Index := 0 TO MAX_IDX_USB_DEV_LIST DO
					gbUSBAvail[Index]										:= bAttachedUSB[Index];
				END_FOR;
			ELSIF ((DevLinkCtrl.FUB.DevLink_0.status <> ERR_FUB_BUSY) AND (DevLinkCtrl.FUB.DevLink_0.status <> ERR_FUB_ENABLE_FALSE)) THEN
				DevLinkCtrl.Step											:= STATE_ERROR_USB;
				DevLinkCtrl.Params.ErrorID									:= DevLinkCtrl.FUB.DevLink_0.status;
				DevLinkCtrl.FUB.DevLink_0.enable							:= FALSE;
			END_IF;
			(* CALL OF FUB *)
			DevLinkCtrl.FUB.DevLink_0();
			(* END OF LINK DEVICE STEP *)

			(* UNLINK DEVICE STEP *)
		STATE_DEV_UNLINK:
			(* SET FUB PARAMS *)
			DevLinkCtrl.FUB.DevUnlink_0.enable	:= TRUE;
			DevLinkCtrl.FUB.DevUnlink_0.handle	:= DevLinkCtrl.Params.FileDevHandle[DevLinkCtrl.Params.Index];

			(* CHECK IF WE HAVE A HANDLE *)
			IF (DevLinkCtrl.Params.FileDevHandle[DevLinkCtrl.Params.Index] = 0) THEN
				DevLinkCtrl.FUB.DevUnlink_0.enable	:= FALSE;
				DevLinkCtrl.Step					:= STATE_WAIT;
			END_IF;

			(* ERROR HANDLING *)
			IF (DevLinkCtrl.FUB.DevUnlink_0.status = ERR_OK) THEN
				DevLinkCtrl.Params.FileDevHandle[DevLinkCtrl.Params.Index]	:= 0;
				DevLinkCtrl.FUB.DevUnlink_0.enable		:= FALSE;
				DevLinkCtrl.Step						:= STATE_WAIT;
			ELSIF ((DevLinkCtrl.FUB.DevUnlink_0.status <> ERR_FUB_BUSY) AND (DevLinkCtrl.FUB.DevUnlink_0.status <> ERR_FUB_ENABLE_FALSE)) THEN
				DevLinkCtrl.Step						:= STATE_ERROR_USB;
				DevLinkCtrl.Params.ErrorID				:= DevLinkCtrl.FUB.DevUnlink_0.status;
				DevLinkCtrl.FUB.DevUnlink_0.enable		:= FALSE;
			END_IF;
			(* CALL OF FUB *)
			DevLinkCtrl.FUB.DevUnlink_0();
			(* END OF UNLINK DEVICE STEP *)

			(* WAIT FOR ERRACK CMD STEP *)
		STATE_ERROR_USB:
			(* DELETE ERROR ID AND GO BACK TO WAIT STEP WHEN ERROR IS ACKNOWLEDGED *)
			IF DevLinkCtrl.Cmd.ErrAck THEN
				DevLinkCtrl.Params.ErrorID	:= 0;
				DevLinkCtrl.Cmd.ErrAck		:= FALSE;
				DevLinkCtrl.Step			:= STATE_WAIT;
			END_IF;
		(* END OF WAIT FOR ERRACK STEP *)
	END_CASE;
	(* END OF STATE MACHINE *)
END_PROGRAM

PROGRAM _EXIT
	(* Insert code here *)
END_PROGRAM
```

### Program Logical/Infrastructure/User/UserMgt (IEC)

#### UserMgt.st - Init, cyclic, exit code
```iecst
//*********************************************************************************
//* Copyright: B&R
//* Author:    B&R
//* Created:   30. Sep 2020/08:00
//* Description: Tasks FOR user control. The User Management handling is done in this task.
//********************************************************************************

PROGRAM _INIT
    // Refresh user data on boot
    User.Command.ListRefresh := TRUE;
END_PROGRAM

PROGRAM _CYCLIC

    IF ArUserInitList_0.ElementName = 'Administrators' THEN
        User.Command.ErrorReset := TRUE;
        User.Command.ListRefresh := TRUE;
    END_IF

    CASE UserManagementState OF

        //*****************Wait For Command************************************************************************************
        IdleUser:
            // Some general UI tasks
            FOR idy := 0 TO (SIZEOF(User.Visualization) / SIZEOF(User.Visualization[0])) - 1 DO
                // --------------------------------------------------------------------------------------------------------------------
                // Create role list for current user
                idx := 0;
                brsmemset(ADR(User.Visualization[idy].ListUserRole), 0, SIZEOF(User.Visualization[idy].ListUserRole));
                WHILE brsstrcmp(ADR(User.Data.Users[User.Visualization[idy].ListUserIndex].Roles[idx]), ADR('')) <> 0 DO
                    String2DataProvider(ADR(User.Data.Users[User.Visualization[idy].ListUserIndex].Roles[idx]), ADR(User.Visualization[idy].ListUserRole[idx]));
                    idx := idx + 1;
                END_WHILE
                // Make sure we dont delete last user role
                IF(idx > 1) THEN
                    User.Visualization[idy].RoleDeleteEnabled := TRUE;
                ELSE
                    User.Visualization[idy].RoleDeleteEnabled := FALSE;
                END_IF
                // Make sure we dont delete last user
                IF(UserCounterTotal[idy] > 0) THEN
                    User.Visualization[idy].UserDeleteEnabled := TRUE;
                ELSE
                    User.Visualization[idy].UserDeleteEnabled := FALSE;
                END_IF
            END_FOR
            // Create new user
            IF  User.Command.UserCreate THEN
                // Make sure passwords match before user is created
                IF((User.Parameter.Password <> '' OR User.Parameter.PasswordRepeat <> '') AND User.Parameter.Password <> User.Parameter.PasswordRepeat) THEN
                    User.Error.No := ERR_PASSWORD_MISMATCH;
                    User.Error.State := UserManagementState;
                    UserManagementState := ErrorUser;
                ELSE
                    tmpUser := User.Parameter.UserName;
                    ArUserCreate_0.Execute := FALSE;
                    UserManagementState := CreateUser;
                END_IF
            ELSIF (User.Command.UserDelete) THEN
                IF(brsstrcmp(ADR(User.Data.UserActive[User.Parameter.VisuSlotID]), ADR(User.Parameter.UserName)) = 0) THEN
                    User.Error.No := ERR_DELETE_CURRENT_USER;
                    User.Error.State := UserManagementState;
                    UserManagementState := ErrorUser;
                ELSE
                    tmpUser := User.Parameter.UserName;
                    ArUserDelete_0.Execute := FALSE;
                    UserManagementState := DeleteUser;
                END_IF
            ELSIF (User.Command.RoleAssign) THEN
                tmpUser := User.Parameter.UserName;
                ArUserAssignRole_0.Execute := FALSE;
                User.Parameter.UserRole := User.Data.Roles[User.Visualization[User.Parameter.VisuSlotID].ListRoleIndex];
                UserManagementState := AssignRole;
                // Remove role from user
            ELSIF (User.Command.RoleRemove) THEN
                tmpUser := User.Parameter.UserName;
                ArUserReleaseRole_0.Execute := FALSE;
                User.Parameter.UserRole := User.Data.Users[User.Visualization[User.Parameter.VisuSlotID].ListUserIndex].Roles[User.Visualization[User.Parameter.VisuSlotID].ListUserRoleIndex];
                UserManagementState := ReleaseRole;
                // Delete user
            ELSIF (User.Command.ListRefresh) THEN
                tmpUser := '';
                UserManagementState := CreateUserListGetFirst;
            ELSIF (User.Command.PasswordChange) THEN
                tmpUser := User.Parameter.UserName;
                ArUserSetPassword_0.Execute := FALSE;
                UserManagementState := ComparePassword;
            ELSIF (User.Command.UserRename) THEN
                // Make sure we dont delete user that is logged in
                IF(brsstrcmp(ADR(User.Data.UserActive[User.Parameter.VisuSlotID]), ADR(User.Parameter.UserName)) = 0) THEN
                    User.Error.No := ERR_RENAME_CURRENT_USER;
                    User.Error.State := UserManagementState;
                    UserManagementState := ErrorUser;
                ELSE
                    tmpUserOld := User.Parameter.UserName;
                    tmpUser := User.Parameter.UserNameNew;
                    ArUserGetProperty_0.Execute := FALSE;
                    ArUserSetProperty_0.Execute := FALSE;
                    ArUserAssignRole_0.Execute := FALSE;
                    ArUserDelete_0.Execute := FALSE;
                    UserManagementState := RenameUser;
                END_IF
            END_IF

            //*****************User Delete************************************************************************************

        DeleteUser:
            ArUserDelete_0.Execute := TRUE;
            ArUserDelete_0.UserName := tmpUser;

            // --------------------------------------------------------------------------------------------------------------------
            // Success
            IF ArUserDelete_0.Done AND NOT ArUserDelete_0.Busy THEN
                // User delete command
                IF User.Command.UserDelete THEN
                    User.Data.Status := 'User >';
                    brsstrcat(ADR(User.Data.Status), ADR(tmpUser));
                    brsstrcat(ADR(User.Data.Status), ADR('< deleted'));
                    // User rename command
                ELSE
                    User.Data.Status := 'User ';
                    brsstrcat(ADR(User.Data.Status), ADR(tmpUserOld));
                    brsstrcat(ADR(User.Data.Status), ADR(' renamed to >'));
                    brsstrcat(ADR(User.Data.Status), ADR(User.Parameter.UserNameNew));
                    brsstrcat(ADR(User.Data.Status), ADR('<'));
                END_IF
                User.Parameter.UserName := '';
                tmpUser := '';
                UserManagementState := CreateUserListGetFirst;
                // Error
            ELSIF ArUserDelete_0.Error THEN
                User.Error.No := ArUserDelete_0.ErrorID;
                User.Error.State := UserManagementState;
                UserManagementState := ErrorUser;
            END_IF
        CreateUser:
            ArUserCreate_0.Execute := TRUE;
            ArUserCreate_0.UserName := tmpUser;

            // --------------------------------------------------------------------------------------------------------------------
            // Success
            IF ArUserCreate_0.Done AND NOT ArUserCreate_0.Busy THEN
                // Create new user
                IF User.Command.UserCreate THEN
                    User.Data.Status := 'User ';
                    brsstrcat(ADR(User.Data.Status), ADR(tmpUser));
                    brsstrcat(ADR(User.Data.Status), ADR(' created'));
                    // Set password when it exists
                    IF User.Parameter.Password <> '' THEN
                        UserManagementState := ComparePassword;
                    ELSE
                        User.Parameter.UserName := '';
                        UserManagementState := CreateUserListGetFirst;
                    END_IF
                    RETURN;
                    // Rename existing user
                ELSE
                    PropertyName := 'UserID';
                    UserManagementState := PropertyRead;
                END_IF
                // Error
            ELSIF ArUserCreate_0.Error THEN
                User.Error.No := ArUserCreate_0.ErrorID;
                User.Error.State := UserManagementState;
                UserManagementState := ErrorUser;
            END_IF
        ComparePassword:
            // --------------------------------------------------------------------------------------------------------------------
            // Success
            IF brsstrcmp(ADR(User.Parameter.Password), ADR(User.Parameter.PasswordRepeat)) = 0 THEN
                UserManagementState := ChangePassword;
                // Error
            ELSE
                User.Error.No := ERR_PASSWORD_MISMATCH;
                User.Error.State := UserManagementState;
                UserManagementState := ErrorUser;
            END_IF
        ChangePassword:
            ArUserSetPassword_0.Execute := TRUE;
            ArUserSetPassword_0.UserName := tmpUser;
            ArUserSetPassword_0.Password := User.Parameter.Password;

            // --------------------------------------------------------------------------------------------------------------------
            // Success
            IF ArUserSetPassword_0.Done AND NOT ArUserSetPassword_0.Busy THEN
                IF User.Command.PasswordChange THEN
                    User.Data.Status := 'Password for user >';
                    brsstrcat(ADR(User.Data.Status), ADR(tmpUser));
                    brsstrcat(ADR(User.Data.Status), ADR('< changed'));
                    User.Parameter.Password := '';
                    User.Parameter.PasswordRepeat := '';
                    User.Command.PasswordChange := FALSE;
                    User.Visualization[User.Parameter.VisuSlotID].ShowMessageBoxOK := TRUE;
                    UserManagementState := IdleUser;
                    RETURN;
                ELSE
                    UserManagementState := CreateUserListGetFirst;
                END_IF
                // Error
            ELSIF ArUserSetPassword_0.Error THEN
                User.Error.No := ArUserSetPassword_0.ErrorID;
                User.Error.State := UserManagementState;
                UserManagementState := ErrorUser;
            END_IF
        CreateUserListGetFirst:
            // Initialize user list
            ArUserInitList_0.Execute := TRUE;
            ArUserInitList_0.ListType := USER_LISTTYPE;
            ArUserInitList_0.ElementName := '';

            // --------------------------------------------------------------------------------------------------------------------
            // Get first user name
            IF ArUserInitList_0.Done AND NOT ArUserInitList_0.Busy THEN

                ArUserGetFirst_0(Execute := TRUE, List := ArUserInitList_0.List);

                // --------------------------------------------------------------------------------------------------------------------
                // Success
                IF ArUserGetFirst_0.Done THEN
                    // Clear data, store user name and generate data provider for vis
                    brsmemset(ADR(User.Data.Users), 0, SIZEOF(User.Data.Users));
                    brsmemset(ADR(User.Visualization[User.Parameter.VisuSlotID].ListUsers), 0, SIZEOF(User.Visualization[User.Parameter.VisuSlotID].ListUsers));
                    brsmemset(ADR(User.Visualization[User.Parameter.VisuSlotID].ListRoles), 0, SIZEOF(User.Visualization[User.Parameter.VisuSlotID].ListRoles));
                    UserCounter := 0;

                    // Make sure user name fits
                    IF(brsstrlen(ADR(ArUserGetFirst_0.ElementName)) < MAX_USER_ITEM_LEN) THEN
                        // Ignore use an anonymous
                        IF ArUserGetFirst_0.ElementName <> 'Anonymous' THEN
                            User.Data.Users[UserCounter].Name := ArUserGetFirst_0.ElementName;
                            String2DataProvider(ADR(ArUserGetFirst_0.ElementName), ADR(User.Visualization[User.Parameter.VisuSlotID].ListUsers[UserCounter]));
                            UserCounter := 1;
                        ELSE
                            UserCounter := 0;
                        END_IF
                        // Reset function block and init counters
                        ArUserGetFirst_0.Execute := FALSE;
                        RoleCounter := 0;
                        UserManagementState := CreateUserListGetNext;
                        // User name is too long
                    ELSE
                        User.Error.No := ERR_USER_ROLE_NAME_SIZE;
                        User.Error.State := UserManagementState;
                        UserManagementState := ErrorUser;
                    END_IF
                    // Error
                ELSIF ArUserGetFirst_0.Error THEN
                    User.Error.No := ArUserGetFirst_0.ErrorID;
                    User.Error.State := UserManagementState;
                    UserManagementState := ErrorUser;
                END_IF
                // Error
            ELSIF ArUserInitList_0.Error THEN
                User.Error.No := ArUserInitList_0.ErrorID;
                User.Error.State := UserManagementState;
                UserManagementState := ErrorUser;
            END_IF
        CreateUserListGetNext:
            // Make sure we have space left
            IF UserCounter < SIZEOF(User.Data.Users)/SIZEOF(User.Data.Users[0]) THEN
                // Get next user

                ArUserGetNext_0(Execute := TRUE,  List := ArUserInitList_0.List);

                // --------------------------------------------------------------------------------------------------------------------
                // Success
                IF ArUserGetNext_0.Done THEN
                    // Make sure user name fits
                    IF(brsstrlen(ADR(ArUserGetNext_0.ElementName)) < MAX_USER_ITEM_LEN) THEN
                        // Ignore use an anonymous
                        IF(ArUserGetNext_0.ElementName <> 'Anonymous') THEN
                            // Store user name and generate data provider for vis
                            User.Data.Users[UserCounter].Name := ArUserGetNext_0.ElementName;
                            String2DataProvider(ADR(ArUserGetNext_0.ElementName), ADR(User.Visualization[User.Parameter.VisuSlotID].ListUsers[UserCounter]));
                            // Reset function block and get next name
                            UserCounter := UserCounter + 1;
                        END_IF
                        ArUserGetNext_0.Execute := FALSE;
                        // User name is too long
                    ELSE
                        User.Error.No := ERR_USER_ROLE_NAME_SIZE;
                        User.Error.State := UserManagementState;
                        UserManagementState := ErrorUser;
                    END_IF
                    // Error
                ELSIF ArUserGetNext_0.Error AND NOT (ArUserGetNext_0.ErrorID = END_OF_LIST) THEN
                    User.Error.No := ArUserGetNext_0.ErrorID;
                    User.Error.State := UserManagementState;
                    UserManagementState := ErrorUser;
                    // List is complete
                ELSIF ArUserGetNext_0.ErrorID = END_OF_LIST THEN
                    // Free up memory
                    ArUserIdent := ArUserInitList_0.List;

                    ArUserDestroyList_0(Execute := TRUE,  List := ArUserIdent);

                    ArUserDestroyList_0(Execute := FALSE,  List := ArUserIdent);

                    // Reset function blocks and counters
                    ArUserGetNext_0.Execute := FALSE;
                    ArUserGetFirst_0.Execute := FALSE;
                    ArUserInitList_0.Execute := FALSE;
                    UserCounterTotal[User.Parameter.VisuSlotID] := UserCounter;
                    UserCounter := 0;
                    RoleCounter := 0;
                    UserManagementState := RoleListInitList;
                END_IF
                // User list is too short
            ELSE
                User.Error.No := ERR_USER_LIST_TOO_SHORT;
                User.Error.State := UserManagementState;
                UserManagementState := ErrorUser;
            END_IF
        RenameUser:
            tmpUserIdx := 0;
            // Find user name in list
            WHILE (brsstrcmp(ADR(User.Data.Users[tmpUserIdx].Name), ADR(tmpUserOld)) <> 0) AND (tmpUserIdx < MAX_USER_NAMES) DO
                tmpUserIdx := tmpUserIdx + 1;
            END_WHILE

            // --------------------------------------------------------------------------------------------------------------------
            // Success
            IF tmpUserIdx < MAX_USER_NAMES THEN
                ArUserCreate_0.Execute := FALSE;
                UserManagementState := CreateUser;
                // Error when user was not found
            ELSE
                User.Error.No := arUSER_ERR_DOES_NOT_EXIST;
                User.Error.State := UserManagementState;
                UserManagementState := ErrorUser;
            END_IF

        RoleListInitList:
            IF User.Data.Users[UserCounter].Name <> '' THEN

                ArUserInitList_0(Execute := TRUE, ListType := USERROLE_LISTTYPE, ElementName := User.Data.Users[UserCounter].Name);

                // --------------------------------------------------------------------------------------------------------------------
                // Success
                IF ArUserInitList_0.Done  AND NOT ArUserInitList_0.Busy THEN

                    ArUserGetFirst_0(Execute := TRUE,  List := ArUserInitList_0.List);
                    // --------------------------------------------------------------------------------------------------------------------
                    // Success
                    IF ArUserGetFirst_0.Done THEN
                        // Make sure role name fits
                        IF(brsstrlen(ADR(ArUserInitList_0.ElementName)) < MAX_USER_ITEM_LEN) THEN
                            User.Data.Users[UserCounter].Roles[0] := ArUserGetFirst_0.ElementName;

                            ArUserGetFirst_0(Execute := FALSE,  List := ArUserInitList_0.List);
                            RoleCounter := 1;
                            UserManagementState := RoleListGetNext;
                            // User role is too long
                        ELSE
                            User.Error.No := ERR_USER_ROLE_NAME_SIZE;
                            User.Error.State := UserManagementState;
                            UserManagementState := ErrorUser;
                        END_IF
                        // Error
                    ELSIF ArUserGetFirst_0.Error THEN
                        User.Error.No := ArUserGetFirst_0.ErrorID;
                        User.Error.State := UserManagementState;
                        UserManagementState := ErrorUser;
                    END_IF
                    // Error
                ELSIF ArUserInitList_0.Error THEN
                    User.Error.No := ArUserInitList_0.ErrorID;
                    User.Error.State := UserManagementState;
                    UserManagementState := ErrorUser;
                END_IF
                // Finish when user roles are complete
            ELSE
                // Reset function blocks
                ArUserInitList_0.Execute := FALSE;
                ArUserGetFirst_0.Execute := FALSE;
                UserCounter := 1;
                RoleCounter := 0;
                UserManagementState := CreateRoleListGetFirst;
            END_IF

        RoleListGetNext:

            ArUserGetNext_0(Execute := TRUE,  List := ArUserInitList_0.List);

            // --------------------------------------------------------------------------------------------------------------------
            // Success
            IF ArUserGetNext_0.Done THEN
                // Make sure user name fits
                IF(brsstrlen(ADR(ArUserGetNext_0.ElementName)) < MAX_USER_ITEM_LEN) THEN
                    User.Data.Users[UserCounter].Roles[RoleCounter] := ArUserGetNext_0.ElementName;
                    RoleCounter := RoleCounter + 1;

                    ArUserGetNext_0(Execute := FALSE,  List := ArUserInitList_0.List);
                    // User role is too long
                ELSE
                    User.Error.No := ERR_USER_ROLE_NAME_SIZE;
                    User.Error.State := UserManagementState;
                    UserManagementState := ErrorUser;
                END_IF
                // List is complete
            ELSIF ArUserGetNext_0.ErrorID = END_OF_LIST THEN
                UserCounter := UserCounter + 1;
                // Free up memory
                ArUserIdent := ArUserInitList_0.List;

                ArUserDestroyList_0(Execute := TRUE,  List := ArUserIdent);

                ArUserDestroyList_0(Execute := FALSE,  List := ArUserIdent);
                // Reset function blocks
                ArUserGetNext_0.Execute := FALSE;
                ArUserInitList_0.Execute := FALSE;
                UserManagementState := RoleListInitList;
                // Error
            ELSIF ArUserGetNext_0.Error THEN
                User.Error.No := ArUserGetNext_0.ErrorID;
                User.Error.State := UserManagementState;
                UserManagementState := ErrorUser;
            END_IF

            // --------------------------------------------------------------------------------------------------------------------
            // Create table of roles
            // --------------------------------------------------------------------------------------------------------------------
        CreateRoleListGetFirst:

            ArUserInitList_0(Execute := TRUE ,ListType := ROLE_LISTTYPE , ElementName := '' );

            // --------------------------------------------------------------------------------------------------------------------
            // Success
            IF ArUserInitList_0.Done AND NOT ArUserInitList_0.Busy THEN

                ArUserGetFirst_0(Execute := TRUE,  List := ArUserInitList_0.List );

                // --------------------------------------------------------------------------------------------------------------------
                // Store role names and generate data provider for vis
                IF ArUserGetFirst_0.Done THEN
                    // Make sure role name fits
                    IF(brsstrlen(ADR(ArUserGetFirst_0.ElementName)) < MAX_USER_ITEM_LEN) THEN
                        User.Data.Roles[RoleCounter] := ArUserGetFirst_0.ElementName;
                        String2DataProvider(ADR(ArUserGetFirst_0.ElementName), ADR(User.Visualization[User.Parameter.VisuSlotID].ListRoles[RoleCounter]));
                        // Reset function block and init counters
                        ArUserGetFirst_0.Execute := FALSE;
                        RoleCounter := 1;
                        UserManagementState := CreateRoleListGetNext;
                        // Role name is too long
                    ELSE
                        User.Error.No := ERR_USER_ROLE_NAME_SIZE;
                        User.Error.State := UserManagementState;
                        UserManagementState := ErrorUser;
                    END_IF
                    // Error
                ELSIF ArUserGetFirst_0.Error THEN
                    User.Error.No := ArUserGetFirst_0.ErrorID;
                    User.Error.State := UserManagementState;
                    UserManagementState := ErrorUser;
                END_IF
                // Error
            ELSIF ArUserInitList_0.Error THEN
                User.Error.No := ArUserInitList_0.ErrorID;
                User.Error.State := UserManagementState;
                UserManagementState := ErrorUser;
            END_IF

        CreateRoleListGetNext:
            IF UserCounter < SIZEOF(User.Data.Roles)/SIZEOF(User.Data.Roles[0]) THEN

                ArUserGetNext_0(Execute := TRUE,  List := ArUserInitList_0.List);

                // --------------------------------------------------------------------------------------------------------------------
                // Store user name and generate data provider for vis
                IF ArUserGetNext_0.Done THEN
                    // Make sure user name fits
                    IF(brsstrlen(ADR(ArUserGetNext_0.ElementName)) < MAX_USER_ITEM_LEN) THEN
                        User.Data.Roles[RoleCounter] := ArUserGetNext_0.ElementName;
                        String2DataProvider(ADR(ArUserGetNext_0.ElementName), ADR(User.Visualization[User.Parameter.VisuSlotID].ListRoles[RoleCounter]));
                        // Reset function block and get next name
                        RoleCounter := RoleCounter + 1;
                        ArUserGetNext_0.Execute := FALSE;
                        // Role name is too long
                    ELSE
                        User.Error.No := ERR_USER_ROLE_NAME_SIZE;
                        User.Error.State := UserManagementState;
                        UserManagementState := ErrorUser;
                    END_IF
                    // Error
                ELSIF ArUserGetNext_0.Error AND NOT (ArUserGetNext_0.ErrorID = END_OF_LIST) THEN
                    User.Error.No := ArUserGetNext_0.ErrorID;
                    User.Error.State := UserManagementState;
                    UserManagementState := ErrorUser;
                    // End of list reached
                ELSIF ArUserGetNext_0.ErrorID = END_OF_LIST THEN
                    // Show message box after succesful command except refresh
                    IF(NOT User.Command.ListRefresh) THEN
                        User.Visualization[User.Parameter.VisuSlotID].ShowMessageBoxOK := TRUE;
                    END_IF
                    // Reset function blocks
                    ArUserGetNext_0.Execute := FALSE;
                    ArUserInitList_0.Execute := FALSE;
                    // Reset function blocks
                    ArUserGetNext_0.Execute := FALSE;
                    ArUserGetFirst_0.Execute := FALSE;
                    ArUserInitList_0.Execute := FALSE;
                    RoleCounter := 0;
                    // Reset command
                    brsmemset(ADR(User.Command), 0, SIZEOF(User.Command));
                    // Select last user if possible
                    IF tmpUser <> '' THEN
                        User.Visualization[User.Parameter.VisuSlotID].ListUserValue := tmpUser;
                    ELSIF(tmpUserNew <> '') THEN
                        User.Visualization[User.Parameter.VisuSlotID].ListUserValue := tmpUserNew;
                    ELSE
                        User.Parameter.UserName := User.Data.Users[0].Name;
                    END_IF
                    // Copy user data into all slots on first boot
                    FOR idy := 0 TO SIZEOF(User.Visualization)/SIZEOF(User.Visualization[0])-1 DO
                        IF(idy <> User.Parameter.VisuSlotID) THEN
                            brsmemcpy(ADR(User.Visualization[idy].ListUsers), ADR(User.Visualization[User.Parameter.VisuSlotID].ListUsers), SIZEOF(User.Visualization[User.Parameter.VisuSlotID].ListUsers));
                            brsmemcpy(ADR(User.Visualization[idy].ListRoles), ADR(User.Visualization[User.Parameter.VisuSlotID].ListRoles), SIZEOF(User.Visualization[User.Parameter.VisuSlotID].ListRoles));
                            UserCounterTotal[idy] := UserCounterTotal[User.Parameter.VisuSlotID];
                        END_IF
                    END_FOR
                    UserManagementState := IdleUser;
                    RETURN;
                END_IF
                // Role list is too short
            ELSE
                User.Error.No := ERR_ROLE_LIST_TOO_SHORT;
                User.Error.State := UserManagementState;
                UserManagementState := ErrorUser;
            END_IF
        PropertyRead:
            ArUserGetProperty_0(Execute := TRUE,  ElementType := arUSER_USER_PROPERTIES, ElementName := tmpUserOld, PropertyName := PropertyName);

            // --------------------------------------------------------------------------------------------------------------------
            // Success
            IF ArUserGetProperty_0.Done AND NOT ArUserGetProperty_0.Busy THEN
                ArUserSetProperty_0.Execute := FALSE;
                UserManagementState := PropertyWrite;
                // Error
            ELSIF ArUserGetProperty_0.Error THEN
                User.Error.No := ArUserGetProperty_0.ErrorID;
                User.Error.State := UserManagementState;
                UserManagementState := ErrorUser;
            END_IF
            // --------------------------------------------------------------------------------------------------------------------
            // Write user property
            // --------------------------------------------------------------------------------------------------------------------
        PropertyWrite:
            ArUserSetProperty_0(Execute := TRUE,  ElementType := arUSER_USER_PROPERTIES, ElementName := tmpUser, PropertyName := PropertyName, PropertyValue := ArUserGetProperty_0.PropertyValue);

            // --------------------------------------------------------------------------------------------------------------------
            // Success
            IF ArUserSetProperty_0.Done AND NOT ArUserSetProperty_0.Busy THEN
                // Read password after user ID
                IF PropertyName = 'UserID' THEN
                    PropertyName := 'Password';
                    ArUserGetProperty_0.Execute := FALSE;
                    UserManagementState := PropertyRead;
                    // Assign roles after password
                ELSIF PropertyName = 'Password' THEN
                    idx := 0;
                    User.Parameter.UserRole := User.Data.Users[tmpUserIdx].Roles[idx];
                    UserManagementState := AssignRole;
                END_IF
                // Error
            ELSIF ArUserSetProperty_0.Error THEN
                User.Error.No := ArUserSetProperty_0.ErrorID;
                User.Error.State := UserManagementState;
                UserManagementState := ErrorUser;
            END_IF

            // --------------------------------------------------------------------------------------------------------------------
        AssignRole:
            ArUserAssignRole_0(Execute := TRUE,  UserName := tmpUser, RoleName := User.Parameter.UserRole);

            // --------------------------------------------------------------------------------------------------------------------
            // Success
            IF User.Command.RoleAssign AND ArUserAssignRole_0.Done AND NOT ArUserAssignRole_0.Busy THEN
                User.Data.Status := 'Role >';
                brsstrcat(ADR(User.Data.Status), ADR(User.Parameter.UserRole));
                brsstrcat(ADR(User.Data.Status), ADR('< assigned to user '));
                brsstrcat(ADR(User.Data.Status), ADR(tmpUser));
                User.Parameter.UserName := '';
                UserManagementState := CreateUserListGetFirst;
            ELSIF User.Command.UserRename AND ((ArUserAssignRole_0.Done AND NOT ArUserAssignRole_0.Busy) OR (ArUserAssignRole_0.ErrorID = arUSER_ERR_ALREADY_EXISTS)) THEN
                idx := idx +1;
                // Assign next role if it exists
                IF User.Data.Users[tmpUserIdx].Roles[idx] <> '' AND idx < MAX_USER_ROLES THEN
                    ArUserAssignRole_0.Execute := FALSE;
                    User.Parameter.UserRole := User.Data.Users[tmpUserIdx].Roles[idx];
                    // Delete old user
                ELSE
                    // Move user names around
                    tmpUserNew := tmpUser;
                    tmpUser := tmpUserOld;
                    UserManagementState := DeleteUser;
                END_IF
                // Error
            ELSIF ArUserAssignRole_0.Error THEN
                User.Error.No := ArUserAssignRole_0.ErrorID;
                User.Error.State := UserManagementState;
                UserManagementState := ErrorUser;
            END_IF

            // --------------------------------------------------------------------------------------------------------------------
            // Release user role
            // --------------------------------------------------------------------------------------------------------------------
        ReleaseRole:
            ArUserReleaseRole_0(Execute := TRUE,  UserName := tmpUser, RoleName := User.Parameter.UserRole);

            // --------------------------------------------------------------------------------------------------------------------
            // Success
            IF ArUserReleaseRole_0.Done AND NOT ArUserReleaseRole_0.Busy THEN
                User.Data.Status := 'Role >';
                brsstrcat(ADR(User.Data.Status), ADR(User.Parameter.UserRole));
                brsstrcat(ADR(User.Data.Status), ADR('< removed from user '));
                brsstrcat(ADR(User.Data.Status), ADR(tmpUser));
                User.Parameter.UserName := '';
                UserManagementState := CreateUserListGetFirst;
                // Error
            ELSIF ArUserReleaseRole_0.Error THEN
                User.Error.No := ArUserReleaseRole_0.ErrorID;
                User.Error.State := UserManagementState;
                UserManagementState := ErrorUser;
            END_IF

        ErrorUser:
            // --------------------------------------------------------------------------------------------------------------------
            // Reset function blocks

            ArUserInitList_0(Execute := FALSE);
            ArUserGetFirst_0(Execute := FALSE);
            ArUserGetNext_0(Execute := FALSE);
            ArUserCreate_0(Execute := FALSE);

            ArUserDelete_0(Execute := FALSE);
            //

            // --------------------------------------------------------------------------------------------------------------------
            // Generate text for most common errors
            IF(User.Error.No = arUSER_ERR_ALREADY_EXISTS) THEN
                User.Error.Text := 'ERR: User/Role already exists or is already assigned';
            ELSIF(User.Error.No = arUSER_ERR_PARAMETER) THEN
                User.Error.Text := 'ERR: User/Role is empty';
            ELSIF(User.Error.No = arUSER_ERR_DOES_NOT_EXIST) THEN
                User.Error.Text := 'ERR: User/Role does not exist';
            ELSIF(User.Error.No = ERR_PASSWORD_MISMATCH) THEN
                User.Error.Text := 'ERR: Passwords do not match';
            ELSIF(User.Error.No = ERR_USER_LIST_TOO_SHORT) THEN
                User.Error.Text := 'ERR: User list is too short';
            ELSIF(User.Error.No = ERR_ROLE_LIST_TOO_SHORT) THEN
                User.Error.Text := 'ERR: Role list is too short';
            ELSIF(User.Error.No = ERR_DELETE_CURRENT_USER) THEN
                User.Error.Text := 'ERR: Can not delete user that is logged in';
            ELSIF(User.Error.No = ERR_USER_ROLE_NAME_SIZE) THEN
                User.Error.Text := 'ERR: User name or role exceeds maximum size of ITEM_LENGTH';
            ELSIF(User.Error.No = ERR_RENAME_CURRENT_USER) THEN
                User.Error.Text := 'ERR: Can not rename user that is logged in';
            ELSE
                User.Error.Text := 'Error executing command';
            END_IF
            // Make sure we dont exceed maximum number of web clients
            IF(User.Parameter.VisuSlotID < SIZEOF(User.Visualization)/SIZEOF(User.Visualization[0])) THEN
                User.Visualization[User.Parameter.VisuSlotID].ShowMessageBoxError := TRUE;
            END_IF
            // --------------------------------------------------------------------------------------------------------------------
            // Return to idle state
            IF User.Command.ErrorReset THEN
                UserCounter := 1;
                RoleCounter := 0;

                brsmemset(ADR(User.Error), 0, SIZEOF(User.Error));
                User.Command.ErrorReset := FALSE;
                User.Visualization[User.Parameter.VisuSlotID].ShowMessageBoxError := FALSE;
                UserManagementState := IdleUser;
            END_IF
            brsmemset(ADR(User.Command), 0, SIZEOF(User.Command));
            RETURN;
        // --------------------------------------------------------------------------------------------------------------------
    END_CASE
    ArUserSetPassword_0();
    ArUserGetNext_0();
    ArUserInitList_0();
    ArUserCreate_0();
    ArUserDelete_0();

    ArUserSetProperty_0();
    ArUserGetProperty_0();
    ArUserAssignRole_0();
    ArUserReleaseRole_0();
    //This instruction Enables the ArUser-Based User Management Page

    gVisuCtrl.cmd.bEnableArUser := TRUE;
    gVisuCtrl.cmd.bEnableMpUserX := FALSE;

    IF X = 1 THEN
        TempStr := "Med is logged in";
        MpAuditCustomEvent(gAuditTrailMpLink, TypeVar, "$$Custom/LoggedIn_ID", TempStr);
    END_IF

END_PROGRAM

PROGRAM _EXIT
	// Insert code here

END_PROGRAM
```

#### UserMgt.typ - Local data types
```iecst
TYPE
	UserParType : 	STRUCT  (*Parameters Data Type for User Management*)
		FilePath : STRING[100];
		UserName : STRING[MAX_USER_ITEM_LEN];
		UserNameNew : STRING[MAX_USER_ITEM_LEN];
		UserRole : STRING[MAX_USER_ITEM_LEN];
		Password : STRING[MAX_USER_ITEM_LEN];
		PasswordRepeat : STRING[MAX_USER_ITEM_LEN];
		VisuSlotID : USINT;
	END_STRUCT;
	UserCmdType : 	STRUCT  (*Command Data Type for User Management*)
		UserCreate : BOOL; (*Create User*)
		UserDelete : BOOL; (*Delete User*)
		UserRename : BOOL; (*Rename User*)
		PasswordChange : BOOL; (*Change Password*)
		RoleAssign : BOOL; (*Assign Role*)
		RoleRemove : BOOL; (*Remove Role*)
		Import : BOOL;
		Export : BOOL;
		ListRefresh : BOOL; (*Refresh List*)
		ErrorReset : BOOL; (*Error Reset*)
	END_STRUCT;
	UserMainType : 	STRUCT  (*Main Control Data Type for User Management*)
		Command : UserCmdType; (*Command of User Management*)
		Parameter : UserParType; (*Parameters for User Management*)
		Data : UserDatType; (*Data for User Management*)
		Visualization : ARRAY[0..MAX_USER_CLIENTS]OF UserVisType; (*Vision related variables for User Management*)
		Error : UserErrType; (*Errors in User Management*)
	END_STRUCT;
	UserDatType : 	STRUCT  (*Data Data Type for User Management*)
		Users : ARRAY[0..MAX_USER_NAMES]OF UserDetailsType; (*Users details*)
		Roles : ARRAY[0..MAX_USER_ROLES]OF STRING[MAX_USER_ITEM_LEN]; (*Roles Details*)
		Status : STRING[200]; (*Status of the user*)
		UserActive : ARRAY[0..MAX_USER_CLIENTS]OF STRING[MAX_USER_ITEM_LEN]; (*Active User*)
	END_STRUCT;
	UserVisType : 	STRUCT  (*User to HMI Data Type for User Management*)
		ListUsers : ARRAY[0..MAX_USER_NAMES]OF STRING[MAX_USER_ITEM_LEN]; (*List of Users*)
		ListUserIndex : UINT; (*List users Index Selection*)
		ListUserValue : STRING[MAX_USER_ITEM_LEN]; (*List User Value*)
		ListUserRole : ARRAY[0..MAX_USER_ROLES]OF STRING[MAX_USER_ITEM_LEN]; (*List User Role*)
		ListUserRoleIndex : UINT; (*List Users Role Index*)
		ListRoles : ARRAY[0..MAX_USER_ROLES]OF STRING[MAX_USER_ITEM_LEN]; (*List Roles*)
		ListRoleIndex : UINT; (*List Roles Index*)
		RoleDeleteEnabled : BOOL; (*Delete Role*)
		UserDeleteEnabled : BOOL; (*User Delete*)
		ShowMessageBoxOK : BOOL; (*Show Message Box*)
		ShowMessageBoxError : BOOL; (*Show Error Message Box*)
	END_STRUCT;
	UserErrType : 	STRUCT  (*Errors Data Type for User Management*)
		No : DINT; (*Error  Numbers*)
		State : UserManagementEnum; (*User Management States*)
		Text : STRING[100]; (*Errors Text*)
	END_STRUCT;
	UserManagementEnum :
		(
		IdleUser, (*Wait state*)
		DestroyList,
		CreateUser,
		DeleteUser,
		RenameUser,
		ExportList,
		ImportList,
		ChangePassword,
		ComparePassword,
		CreateUserListGetNext,
		CreateUserListGetFirst,
		AssignRole,
		ReleaseRole,
		RoleListMain,
		RoleListDeleteList,
		RoleListInitList,
		CreateRoleListGetFirst,
		CreateRoleListGetNext,
		RoleListGetNext,
		PropertyRead,
		PropertyWrite,
		ErrorUser
		);
	UserDetailsType : 	STRUCT
		Roles : ARRAY[0..MAX_USER_ROLES]OF STRING[MAX_USER_ITEM_LEN]; (*User Roles*)
		Name : STRING[MAX_USER_ITEM_LEN]; (*User Names*)
	END_STRUCT;
END_TYPE
```

#### UserMgt.var - Local variables
```iecst
(*ARUser Function Block*)
VAR
	ArUserAssignRole_0 : ArUserAssignRole;
	ArUserCreate_0 : ArUserCreate;
	ArUserDelete_0 : ArUserDelete;
	ArUserDestroyList_0 : ArUserDestroyList;
	ArUserGetFirst_0 : ArUserGetFirst;
	ArUserGetNext_0 : ArUserGetNext;
	ArUserGetProperty_0 : ArUserGetProperty;
	ArUserIdent : ArUserIdentType;
	ArUserInitList_0 : ArUserInitList;
	ArUserReleaseRole_0 : ArUserReleaseRole;
	ArUserSetPassword_0 : ArUserSetPassword;
	UserManagementState : UserManagementEnum;
	ArUserSetProperty_0 : ArUserSetProperty;
END_VAR
(*User Management Variables*)
VAR
	User : UserMainType; (*User Declaration Variable*)
	DataProvider : ARRAY[0..19] OF WSTRING[80] := ["{'value':'4','text':'Entry1'}",19("")];
	Password : WSTRING[80]; (*Password*)
	UserName : WSTRING[80]; (*User Name*)
	tmpUserNew : STRING[MAX_USER_ITEM_LEN];
	tmpUser : STRING[MAX_USER_ITEM_LEN];
	tmpUserOld : STRING[MAX_USER_ITEM_LEN];
	PropertyName : STRING[100]; (*Name of the property*)
	idx : INT; (*Index used for FOR Loop*)
	idy : USINT; (*Index used for FOR Loop*)
	UserCounter : USINT;
	tmpUserIdx : USINT; (*Index used for FOR Loop*)
	RoleCounter : USINT;
	UserCounterTotal : ARRAY[0..MAX_USER_CLIENTS] OF USINT;
	NewUserName : WSTRING[20];
	NewUserConfirmPassword : WSTRING[20];
	NewUserPassword : WSTRING[20];
	CreateNewUser : BOOL;
	TempStr : WSTRING[100];
	TypeVar : WSTRING[100];
	X : BOOL;
	Status : DINT;
END_VAR
(*Constants*)
VAR CONSTANT
	ROLE_LISTTYPE : BYTE := 2; (*List Type Role*)
	USERROLE_LISTTYPE : BYTE := 3; (*List Type UserRole*)
	USER_LISTTYPE : BYTE := 1; (*List Type User*)
	MAX_USER_ROLES : USINT := 20; (*Maximum number of user roles*)
	MAX_USER_NAMES : USINT := 50; (*Maximum number of users*)
	MAX_USER_CLIENTS : USINT := 2; (*Maximum number of concurrent web clients*)
	MAX_USER_ITEM_LEN : USINT := 60; (*String length for users and roles*)
	ERR_PASSWORD_MISMATCH : DINT := 50000; (*Passwords dont match*)
	ERR_USER_LIST_TOO_SHORT : DINT := 50001; (*More users found than fit into user list*)
	ERR_ROLE_LIST_TOO_SHORT : DINT := 50002; (*More roles found than fit into the role list*)
	ERR_DELETE_CURRENT_USER : DINT := 50003; (*Logged in user can not be deleted*)
	ERR_RENAME_CURRENT_USER : DINT := 50004; (*Logged in user can not be renamed*)
	ERR_USER_ROLE_NAME_SIZE : DINT := 50005; (*Logged in user can not be renamed*)
	ERR_USER_TOO_MANY_CLIENTS : DINT := 50010; (*More than 3 clients try to connect to user managment*)
	END_OF_LIST : DINT := -2144327714; (*End of list reached*)
END_VAR
```

#### LocalFunctions.fun
```iecst
{REDUND_ERROR} FUNCTION String2DataProvider : BOOL (*TODO: Add your comment here*) (*$GROUP=User,$CAT=User,$GROUPICON=User.png,$CATICON=User.png*)
	VAR_INPUT
		SourceString : UDINT;
		TargetString : UDINT;
	END_VAR
END_FUNCTION
```

#### LocalFunctions.st
```iecst
// --------------------------------------------------------------------------------------------------------------------
// Create mappView data provider string
FUNCTION String2DataProvider
	brsstrcpy(TargetString, ADR('{"value":"'));
	brsstrcat(TargetString, SourceString);
	brsstrcat(TargetString, ADR('","text":"'));
	brsstrcat(TargetString, SourceString);
	brsstrcat(TargetString, ADR('"}'));
	String2DataProvider := TRUE;
END_FUNCTION
```

### Package Logical/MainControl - Package Cross Cutter Control

### Program Logical/MainControl/MainCtrl

#### Types.typ
```iecst
TYPE
	AxisStateEnum :
		(
		AX_STATE_WAIT := 0,
		AX_STATE_POWER_ON,
		AX_STATE_HOME,
		AX_STATE_READY,
		AX_STATE_STOP,
		AX_STATE_JOG_POSITIVE,
		AX_STATE_JOG_NEGATIVE,
		AX_STATE_MOVE_ABSOLUTE,
		AX_STATE_MOVE_ADDITIVE,
		AX_STATE_MOVE_VELOCITY,
		AX_STATE_HALT,
		AX_STATE_TORQUE_CONTROL,
		AX_STATE_CAM_AUTOMAT,
		AX_STATE_ERROR := 90,
		AX_STATE_ERROR_RESET
		);
	AxControlCommandType : 	STRUCT  (*command structure*)
		Power : BOOL; (*switch on the controller*)
		Home : BOOL; (*reference the axis*)
		MoveAbsolute : BOOL; (*move to an defined position*)
		MoveAdditive : BOOL; (*move a defiened distance*)
		MoveVelocity : BOOL; (*start a movement with a defiened velocity*)
		MoveJogPos : BOOL; (*move in positive direction as long as is set*)
		MoveJogNeg : BOOL; (*move in negative direction as long as is set*)
		TorqueControl : BOOL; (*Activate torque limitation*)
		Stop : BOOL; (*stop every active movement as long as is set*)
		RunCamAutomat : BOOL; (*start coupling beetween master and slave*)
		ErrorAcknowledge : BOOL; (*reset active errors*)
		Reset : BOOL;
	END_STRUCT;
	AxControlParameterType : 	STRUCT  (*parameter structure*)
		AxPar : MpAxisBasicParType; (*Cutter axis parameters*)
	END_STRUCT;
	AxControlStatusType : 	STRUCT  (*status structure*)
		ErrorID : UDINT; (*ErrorID of any occured error*)
		Error : BOOL; (*Error on MpAxisBasic*)
		ActPosition : LREAL; (*actual position of the axis [mm OR °]*)
		ActVelocity : LREAL; (*actual velocity of the axis [mm/s OR °]*)
		ActTorque : REAL; (*actual torque [Nm]*)
		ActualPLCOpenState : McAxisPLCopenStateEnum; (*actual PLCopen state*)
		TorqueLimited : BOOL; (*Torque is currently being limited*)
		MovementActive : BOOL; (*A movement is currently active*)
		PowerOn : BOOL; (*Axis is powered on*)
		IsHomed : BOOL; (*Axis is homed*)
	END_STRUCT;
	AxControlType : 	STRUCT  (*control structure*)
		Command : AxControlCommandType; (*command structure*)
		Parameter : AxControlParameterType; (*parameter structure*)
		Status : AxControlStatusType; (*status structure*)
		AxisState : AxisStateEnum;
	END_STRUCT;
END_TYPE

(*Main Control*)

TYPE
	MainStatusType : 	STRUCT  (*Structure Type for Main Control Status*)
		MachineStatus : STRING[80]; (*Machine Status*)
		CurrentBatch : INT; (*Cutting Batch Index*)
		CuttingProcessFinished : BOOL; (*Cutting process Finished*)
		BatchIdxCutNumber : INT; (*Batch Index Cut Number*)
		CuttingCycle : INT; (*Cutting Cycle*)
		ProductsCutTotal : UINT;
		ProductsCutBatch : UINT; (*Product Cut Numbebr*)
		CurrentBatchLength : REAL; (*Current batch product length [mm]*)
		CurrentBatchTarget : UINT; (*Current batch production target*)
	END_STRUCT;
	MainCmdType : 	STRUCT  (*Structure Type for Main Control Commands*)
		AutoModeOn : BOOL; (*Power on axes*)
		RunFeeder : BOOL; (*Run the process*)
		RunCutter : BOOL; (*Homing of the Axis*)
	END_STRUCT;
	MainFixParametersType : 	STRUCT
		MinProductLength : REAL := 50; (*Minimum product length [mm]*)
		MaxProductLength : REAL := 1000; (*Maximum product length [mm]*)
		SyncAngle : REAL := 20; (*Sync Angle [°]*)
		NrOfKnives : USINT := 1; (*Number of knives*)
		CutDiameter : REAL := 90; (*Cutter radius [mm]*)
	END_STRUCT;
	MainParametersType : 	STRUCT
		ProductNumber : ARRAY[0..4]OF INT; (*Product Number*)
		ProductLength : ARRAY[0..4]OF REAL; (*Real Product Length*)
		AxPar : ARRAY[0..MAX_IDX_AXIS]OF MpAxisBasicParType; (*Axis parameters*)
	END_STRUCT;
	MainInternType : 	STRUCT  (*Structure Type for Main Control Parameters*)
		ProductNumber : ARRAY[0..4]OF UINT; (*Product Number*)
		ProductLength : ARRAY[0..4]OF REAL; (*Real Product Length*)
	END_STRUCT;
	MainCtrlType : 	STRUCT  (*Structure Type for Main Control *)
		Command : MainCmdType; (*Main Control Command*)
		FixParameter : MainFixParametersType; (*Main Control Parameters*)
		Parameter : MainParametersType; (*Main Control Parameters*)
		Status : MainStatusType; (*Main Control Status*)
		Intern : MainInternType;
	END_STRUCT;
END_TYPE
```

#### Variables.var
```iecst
(*Main Control----------------------------------------*)
VAR
	MainCtrl : MainCtrlType; (*Main Control Variable*)
	MpAxisBasic_x : ARRAY[0..MAX_IDX_AXIS] OF MpAxisBasic; (*MpAxis Declaration*)
	PreviewParameters : MainParametersType;
	MpRecipeRegPar_M : MpRecipeRegPar; (*Register fix parameters to MpRecipe*)
	MpRecipeRegPar_Pre1 : MpRecipeRegPar; (*Register preview parameters*)
	MpRecipeRegPar_Pre2 : MpRecipeRegPar; (*Register preview parameters*)
	MpRecipeRegPar_P : MpRecipeRegPar; (*Register product parameters to MpRecipe*)
	ReactionName : STRING[80]; (*String to check for MpAlarmX reactions*)
	LastAutoModeOn : BOOL; (*Last cycle's status of auto mode on switch*)
	ResetEditValues : BOOL;
	CopyPreviewParameters : BOOL;
END_VAR
(*Motion Control Related Variables ------------------------------------------------------------------------------------------------*)
VAR
	AxisControl : ARRAY[0..MAX_IDX_AXIS] OF AxControlType; (*control structure*)
	McCamAutDefine : McAcpAxCamAutDefineType; (*Definition of cam automat parameters*)
	McCamAutPar : McAcpAxCamAutParType; (*Cam automat parameters*)
	MC_ReadAxisError_x : ARRAY[0..MAX_IDX_AXIS] OF MC_ReadAxisError; (*Read Axis Error Function Block*)
	MC_ReadActualTorque_x : ARRAY[0..MAX_IDX_AXIS] OF MC_ReadActualTorque; (*Read Actual PositionFunction Block *)
	MC_BR_CamAutomatCommand_0 : MC_BR_CamAutomatCommand; (*Cam Automat Command Function Block*)
	MC_BR_CamAutomatGetPar_AcpAx_0 : MC_BR_CamAutomatGetPar_AcpAx; (*Get Cam Automat Parameters Function Block*)
	MC_BR_CamAutomatSetPar_AcpAx_0 : MC_BR_CamAutomatSetPar_AcpAx; (*Set Cam Automat Parameters Function Block*)
	StopMovementsReaction : BOOL; (*Stop movements on positive edge of alarm reaction*)
	AxIndex : USINT := 0; (*Index for Axis in FOR Statement*)
	InitCamAut : USINT; (*state of initializing camaut data*)
	UpdateCamAutomat : BOOL;
	CamUpdateState : USINT;
END_VAR
(*Constants---------------------------------------------------------------------------------------------------------------------------------*)
VAR CONSTANT
	AXIS_IDX_FEEDER : USINT := 0; (*Axis index of the feeder axis*)
	AXIS_IDX_CUTTER : USINT := 1; (*Axis index of the cutter axis*)
	MAX_IDX_AXIS : USINT := 1; (*Max axis index*)
END_VAR
```

#### AxisStateMachine.st
```iecst
//*********************************************************************************
//* Copyright: B&R Industrial Automation GmbH
//* Created:   28 June, 2021/14:13
//* This file contains the logic to control an axis
//*********************************************************************************

ACTION AxisStateMachine:
	StopMovementsReaction := EDGEPOS(MpAlarmXCheckReaction(gMpLinkAlarmXCore, 'StopMovements'));
	FOR AxIndex := 0 TO MAX_IDX_AXIS DO
		// Update parameters on recipe load
		IF MpRecipeRegPar_P.UpdateNotification THEN
			brsmemcpy(ADR(AxisControl[AxIndex].Parameter.AxPar), ADR(MainCtrl.Parameter.AxPar[AxIndex]), SIZEOF(AxisControl[AxIndex].Parameter.AxPar));
		END_IF

		CASE AxisControl[AxIndex].AxisState OF

			AX_STATE_WAIT: // Wait for command
				IF AxisControl[AxIndex].Command.Home THEN
					AxisControl[AxIndex].Parameter.AxPar.Homing.Mode := mcHOMING_DEFAULT;
					MpAxisBasic_x[AxIndex].Home := TRUE;
					IF NOT MpAxisBasic_x[AxIndex].IsHomed THEN
						AxisControl[AxIndex].AxisState := AX_STATE_HOME;
					END_IF
				ELSIF AxisControl[AxIndex].Command.MoveJogPos THEN
//					MpAxisBasic_x[AxIndex].JogPositive := TRUE;
					MpAxisBasic_x[AxIndex].MoveVelocity := TRUE;
					AxisControl[AxIndex].Parameter.AxPar.Direction := mcDIR_POSITIVE;
					AxisControl[AxIndex].AxisState := AX_STATE_JOG_POSITIVE;
				ELSIF AxisControl[AxIndex].Command.MoveJogNeg THEN
//					MpAxisBasic_x[AxIndex].JogNegative := TRUE;
					MpAxisBasic_x[AxIndex].MoveVelocity := TRUE;
					AxisControl[AxIndex].Parameter.AxPar.Direction := mcDIR_NEGATIVE;
					AxisControl[AxIndex].AxisState := AX_STATE_JOG_NEGATIVE;
				ELSIF AxisControl[AxIndex].Command.MoveAbsolute THEN
					AxisControl[AxIndex].Parameter.AxPar.Direction := mcDIR_SHORTEST_WAY;
					MpAxisBasic_x[AxIndex].MoveAbsolute := TRUE;
					AxisControl[AxIndex].AxisState := AX_STATE_MOVE_ABSOLUTE;
				ELSIF AxisControl[AxIndex].Command.MoveAdditive THEN
					MpAxisBasic_x[AxIndex].MoveAdditive := TRUE;
					AxisControl[AxIndex].AxisState := AX_STATE_MOVE_ADDITIVE;
				ELSIF AxisControl[AxIndex].Command.MoveVelocity THEN
					AxisControl[AxIndex].Parameter.AxPar.Direction := mcDIR_POSITIVE;
					MpAxisBasic_x[AxIndex].MoveVelocity := TRUE;
					AxisControl[AxIndex].AxisState := AX_STATE_MOVE_VELOCITY;
				ELSIF AxisControl[AxIndex].Command.RunCamAutomat THEN
					AxisControl[AxIndex].AxisState := AX_STATE_CAM_AUTOMAT;
				END_IF

			AX_STATE_HOME:
				IF MpAxisBasic_x[AxIndex].IsHomed THEN
					// Homing done
					AxisControl[AxIndex].Command.Home := FALSE;
					MpAxisBasic_x[AxIndex].Home := FALSE;
					AxisControl[AxIndex].AxisState := AX_STATE_WAIT;
				ELSIF (NOT AxisControl[AxIndex].Command.Home) OR AxisControl[AxIndex].Command.Stop THEN
					// Homing canceled or stopped
					AxisControl[AxIndex].Command.Home := FALSE;
					AxisControl[AxIndex].Command.Stop := FALSE;
					MpAxisBasic_x[AxIndex].Home := FALSE;
					AxisControl[AxIndex].AxisState := AX_STATE_WAIT;
				END_IF

			AX_STATE_JOG_POSITIVE:
				IF (NOT AxisControl[AxIndex].Command.MoveJogPos) OR AxisControl[AxIndex].Command.Stop THEN
					// Jog done or stopped
//					MpAxisBasic_x[AxIndex].JogPositive := FALSE;
					AxisControl[AxIndex].Command.MoveJogPos := FALSE;
					AxisControl[AxIndex].Command.Stop := FALSE;
					MpAxisBasic_x[AxIndex].MoveVelocity := FALSE;
					AxisControl[AxIndex].AxisState := AX_STATE_WAIT;
				END_IF

			AX_STATE_JOG_NEGATIVE:
				IF (NOT AxisControl[AxIndex].Command.MoveJogNeg) OR AxisControl[AxIndex].Command.Stop THEN
					// Jog done or stopped
//					MpAxisBasic_x[AxIndex].JogPositive := FALSE;
					AxisControl[AxIndex].Command.MoveJogNeg := FALSE;
					AxisControl[AxIndex].Command.Stop := FALSE;
					MpAxisBasic_x[AxIndex].MoveVelocity := FALSE;
					AxisControl[AxIndex].AxisState := AX_STATE_WAIT;
				END_IF

			AX_STATE_MOVE_ABSOLUTE:
				IF NOT AxisControl[AxIndex].Command.MoveAbsolute OR MpAxisBasic_x[AxIndex].MoveDone OR AxisControl[AxIndex].Command.Stop THEN
					// Move absolut done or stopped
					MpAxisBasic_x[AxIndex].MoveAbsolute := FALSE;
					AxisControl[AxIndex].Command.Stop := FALSE;
					AxisControl[AxIndex].Command.MoveAbsolute := FALSE;
					AxisControl[AxIndex].AxisState := AX_STATE_WAIT;
				END_IF

			AX_STATE_MOVE_ADDITIVE:
				// Move additive done or stopped
				IF NOT AxisControl[AxIndex].Command.MoveAdditive OR MpAxisBasic_x[AxIndex].MoveDone OR AxisControl[AxIndex].Command.Stop THEN
					MpAxisBasic_x[AxIndex].MoveAdditive := FALSE;
					AxisControl[AxIndex].Command.Stop := FALSE;
					AxisControl[AxIndex].Command.MoveAdditive := FALSE;
					AxisControl[AxIndex].AxisState := AX_STATE_WAIT;
				END_IF

			AX_STATE_MOVE_VELOCITY:
				IF (NOT AxisControl[AxIndex].Command.MoveVelocity) OR AxisControl[AxIndex].Command.Stop THEN
					// Move velocity done or stopped
					AxisControl[AxIndex].Command.MoveVelocity := FALSE;
					AxisControl[AxIndex].Command.Stop := FALSE;
					MpAxisBasic_x[AxIndex].MoveVelocity := FALSE;
					AxisControl[AxIndex].AxisState := AX_STATE_WAIT;
				END_IF

			AX_STATE_CAM_AUTOMAT:
				// Start synchronized movement
				IF MC_BR_CamAutomatCommand_0.Ready THEN
					MC_BR_CamAutomatCommand_0.Start := AxisControl[AxIndex].Command.RunCamAutomat AND NOT MC_BR_CamAutomatCommand_0.Running;
				END_IF
				// Stop synchronized movement
				IF (NOT AxisControl[AxIndex].Command.RunCamAutomat) OR AxisControl[AxIndex].Command.Stop THEN
					AxisControl[AxIndex].Command.RunCamAutomat := FALSE;
					AxisControl[AxIndex].Command.Stop := FALSE;
					MC_BR_CamAutomatCommand_0.EndAutomat := MC_BR_CamAutomatCommand_0.Running;
					IF NOT MC_BR_CamAutomatCommand_0.Running THEN
						// Automat has stopped
						AxisControl[AxIndex].AxisState := AX_STATE_WAIT;
					END_IF
				END_IF

			AX_STATE_ERROR:
				// Stop movements and reset .Power input if power is lost
				AxisControl[AxIndex].Command.Home := FALSE;
				AxisControl[AxIndex].Command.MoveAbsolute := FALSE;
				AxisControl[AxIndex].Command.MoveAdditive := FALSE;
				AxisControl[AxIndex].Command.MoveJogNeg := FALSE;
				AxisControl[AxIndex].Command.MoveJogPos := FALSE;
				AxisControl[AxIndex].Command.MoveVelocity := FALSE;
				AxisControl[AxIndex].Command.RunCamAutomat := FALSE;
				MpAxisBasic_x[AxIndex].Home := FALSE;
				MpAxisBasic_x[AxIndex].JogNegative := FALSE;
				MpAxisBasic_x[AxIndex].JogPositive := FALSE;
				MpAxisBasic_x[AxIndex].MoveVelocity := FALSE;
				MpAxisBasic_x[AxIndex].MoveAbsolute := FALSE;
				MpAxisBasic_x[AxIndex].MoveAdditive := FALSE;
				MpAxisBasic_x[AxIndex].Power := MpAxisBasic_x[AxIndex].PowerOn AND AxisControl[AxIndex].Command.Power;
				MC_BR_CamAutomatCommand_0.Start := FALSE;
				MC_BR_CamAutomatCommand_0.Stop := MC_BR_CamAutomatCommand_0.Running;
				IF NOT MpAxisBasic_x[AxIndex].MoveActive AND NOT MC_BR_CamAutomatCommand_0.Running THEN
					// Wait for error acknowledge
					IF AxIndex = 0 THEN
						brsstrcpy(ADR(ReactionName), ADR('MasterWaitAcknowledge'));
					ELSIF AxIndex = 1 THEN
						brsstrcpy(ADR(ReactionName), ADR('SlaveWaitAcknowledge'));
					END_IF
					IF AxisControl[AxIndex].Command.ErrorAcknowledge OR NOT MpAlarmXCheckReaction(gMpLinkAlarmXCore, ReactionName)  THEN
						AxisControl[AxIndex].Command.ErrorAcknowledge := FALSE;
						AxisControl[AxIndex].AxisState := AX_STATE_ERROR_RESET;
					END_IF
				END_IF

			AX_STATE_ERROR_RESET:
				// Check if CamAutomat needs to be reset
				MC_BR_CamAutomatCommand_0.Enable := NOT MC_BR_CamAutomatCommand_0.Error AND NOT MC_BR_CamAutomatCommand_0.CommandAborted;

				// Reset MpAxisBasic errors
				MpAxisBasic_x[AxIndex].ErrorReset := MpAxisBasic_x[AxIndex].Error;
				MpAxisBasic_x[AxIndex].Power := MpAxisBasic_x[AxIndex].PowerOn AND AxisControl[AxIndex].Command.Power;

				// Back to wait state when errors are reset
				IF NOT MpAxisBasic_x[AxIndex].Error AND NOT MC_BR_CamAutomatCommand_0.Error AND MC_BR_CamAutomatCommand_0.Valid THEN
					AxisControl[AxIndex].AxisState := AX_STATE_WAIT;
				END_IF
		END_CASE;

		// Reset stop command when axis is not moving
		IF NOT MpAxisBasic_x[AxIndex].MoveActive OR MpAxisBasic_x[AxIndex].Stopped THEN
			AxisControl[AxIndex].Command.Stop := FALSE;
		END_IF

		// Check alarm reaction
		IF StopMovementsReaction THEN
			AxisControl[AxIndex].Command.Home := FALSE;
			AxisControl[AxIndex].Command.MoveAbsolute := FALSE;
			AxisControl[AxIndex].Command.MoveAdditive := FALSE;
			AxisControl[AxIndex].Command.MoveJogNeg := FALSE;
			AxisControl[AxIndex].Command.MoveJogPos := FALSE;
			AxisControl[AxIndex].Command.MoveVelocity := FALSE;
			AxisControl[AxIndex].Command.RunCamAutomat := FALSE;
			AxisControl[AxIndex].Command.Stop := MpAxisBasic_x[AxIndex].MoveActive;
		END_IF

		// Reset power command if not ready to power on
		IF NOT MpAxisBasic_x[AxIndex].Info.ReadyToPowerOn THEN
			AxisControl[AxIndex].Command.Power := FALSE;
		END_IF

		// Always directly access power, stop, and torque control
		IF AxisControl[AxIndex].AxisState < AX_STATE_ERROR THEN
			MpAxisBasic_x[AxIndex].Power := AxisControl[AxIndex].Command.Power;
			MpAxisBasic_x[AxIndex].Stop := AxisControl[AxIndex].Command.Stop;
			MpAxisBasic_x[AxIndex].LimitLoad := AxisControl[AxIndex].Command.TorqueControl AND MpAxisBasic_x[AxIndex].PowerOn AND MpAxisBasic_x[AxIndex].IsHomed;
		END_IF

		// Reset update command when update is done, or no movement is active
		IF MpAxisBasic_x[AxIndex].UpdateDone OR NOT MpAxisBasic_x[AxIndex].MoveActive THEN
			MpAxisBasic_x[AxIndex].Update := FALSE;
		END_IF
	END_FOR
END_ACTION
```

#### AxisStatusUpdate.st
```iecst
//*********************************************************************************
//* Copyright: B&R Industrial Automation GmbH
//* Created:   29 June, 2021/09:58
//* This file contains the logic to update the axis status information
//*********************************************************************************

ACTION AxisStatusUpdate:
	FOR AxIndex := 0 TO MAX_IDX_AXIS DO
		//*********************** MpAxisBasic_x information ************************
		AxisControl[AxIndex].Status.ActualPLCOpenState := MpAxisBasic_x[AxIndex].Info.PLCopenState;
		AxisControl[AxIndex].Status.MovementActive := MpAxisBasic_x[AxIndex].MoveActive;
		AxisControl[AxIndex].Status.TorqueLimited := MpAxisBasic_x[AxIndex].Info.LimitLoadActive;
		AxisControl[AxIndex].Status.ActPosition := MpAxisBasic_x[AxIndex].Position;
		AxisControl[AxIndex].Status.ActVelocity := MpAxisBasic_x[AxIndex].Velocity;
		AxisControl[AxIndex].Status.Error := MpAxisBasic_x[AxIndex].Error;
		AxisControl[AxIndex].Status.PowerOn := MpAxisBasic_x[AxIndex].PowerOn;
		AxisControl[AxIndex].Status.IsHomed := MpAxisBasic_x[AxIndex].IsHomed;

		IF MpAxisBasic_x[AxIndex].Active AND (MpAxisBasic_x[AxIndex].Info.CommunicationState = mcCOMM_STATE_ACTIVE) THEN
			//******************* MC_READACTUALTORQUE ********************
			MC_ReadActualTorque_x[AxIndex].Enable := NOT(MC_ReadActualTorque_x[AxIndex].Error);
			MC_ReadActualTorque_x[AxIndex]();
			IF MC_ReadActualTorque_x[AxIndex].Valid THEN
				AxisControl[AxIndex].Status.ActTorque := MC_ReadActualTorque_x[AxIndex].Torque;
			END_IF

			//*********************** MC_READAXISERROR *********************
			MC_ReadAxisError_x[AxIndex].Enable := NOT(MC_ReadAxisError_x[AxIndex].Error);
			MC_ReadAxisError_x[AxIndex]();
			IF MC_ReadAxisError_x[AxIndex].Valid THEN
				AxisControl[AxIndex].Status.ErrorID := MC_ReadAxisError_x[AxIndex].AxisErrorID;
			END_IF
		END_IF

		//*************** CHECK FOR GENERAL AXIS ERROR *****************
		IF ((MC_ReadAxisError_x[AxIndex].AxisErrorID <> 0) AND MC_ReadAxisError_x[AxIndex].Valid) OR MpAxisBasic_x[AxIndex].Error THEN
			// Set error state if not already in error state / or error reset state
			IF AxisControl[AxIndex].AxisState < AX_STATE_ERROR THEN
				AxisControl[AxIndex].AxisState := AX_STATE_ERROR;
			END_IF
		ELSIF AxisControl[AxIndex].AxisState < AX_STATE_ERROR THEN
			AxisControl[AxIndex].Command.ErrorAcknowledge := FALSE ;
		END_IF
	END_FOR // FOR uAxIndex := 0 TO MAX_IDX_AXIS DO
END_ACTION
```
